METHOD PRIVATE M_Manual_Cylinder
VAR_INPUT
END_VAR
CylinderManualCtrl[1](bTrigger:=StorageManualCommand.UpCV.FeedInPress1.Exetend);
CylinderManualCtrl[2](bTrigger:=StorageManualCommand.UpCV.FeedInPress2.Exetend);
CylinderManualCtrl[3](bTrigger:=StorageManualCommand.UpCV.DiameterPress.Exetend);
CylinderManualCtrl[4](bTrigger:=StorageManualCommand.UpCV.CamaraPress1.Exetend);
CylinderManualCtrl[5](bTrigger:=StorageManualCommand.UpCV.CamaraPress2.Exetend);
CylinderManualCtrl[6](bTrigger:=StorageManualCommand.UpCV.CamaraPress3.Exetend);
CylinderManualCtrl[7](bTrigger:=StorageManualCommand.UpCV.CamaraPress4.Exetend);
CylinderManualCtrl[8](bTrigger:=StorageManualCommand.UpCV.Block1.Exetend);
CylinderManualCtrl[9](bTrigger:=StorageManualCommand.UpCV.Block2.Exetend);
CylinderManualCtrl[10](bTrigger:=StorageManualCommand.UpCV.Block3.Exetend);
CylinderManualCtrl[11](bTrigger:=StorageManualCommand.UpCV.DiameterHoriz.Exetend);
CylinderManualCtrl[12](bTrigger:=StorageManualCommand.UpCV.DiameterVert.Exetend);
CylinderManualCtrl[13](bTrigger:=StorageManualCommand.UpCV.DiameterClamp.Exetend);
CylinderManualCtrl[14](bTrigger:=StorageManualCommand.UpCV.StackPush.Exetend);
CylinderManualCtrl[15](bTrigger:=AllocateManualCommand.PullOutCV.AsidePress1.Exetend);
CylinderManualCtrl[16](bTrigger:=AllocateManualCommand.PullOutCV.AsidePress2.Exetend);
CylinderManualCtrl[17](bTrigger:=AllocateManualCommand.PullOutCV.AsideBlock.Exetend);
CylinderManualCtrl[18](bTrigger:=AllocateManualCommand.PullOutCV.BsidePress1.Exetend);
CylinderManualCtrl[19](bTrigger:=AllocateManualCommand.PullOutCV.BsidePress2.Exetend);
CylinderManualCtrl[20](bTrigger:=AllocateManualCommand. PullOutCV.BsideBlock.Exetend);
CylinderManualCtrl[21](bTrigger:=StorageManualCommand.LowCV.Press1.Exetend);
CylinderManualCtrl[22](bTrigger:=StorageManualCommand.LowCV.Press2.Exetend);
CylinderManualCtrl[23](bTrigger:=StorageManualCommand.LowCV.Press3.Exetend);
CylinderManualCtrl[24](bTrigger:=StorageManualCommand.LowCV.Press4.Exetend);
CylinderManualCtrl[25](bTrigger:=StorageManualCommand.LowCV.Block1.Exetend);
CylinderManualCtrl[26](bTrigger:=StorageManualCommand.LowCV.Block2.Exetend);
CylinderManualCtrl[27](bTrigger:=AllocateManualCommand.AllocatedRobot.LeftVert1.Exetend);
CylinderManualCtrl[28](bTrigger:=AllocateManualCommand.AllocatedRobot.LeftVert2.Exetend);
CylinderManualCtrl[29](bTrigger:=AllocateManualCommand.AllocatedRobot.RightVert1.Exetend);
CylinderManualCtrl[30](bTrigger:=AllocateManualCommand.AllocatedRobot.RightVert2.Exetend);
CylinderManualCtrl[31](bTrigger:=AllocateManualCommand.AllocatedRobot.LeftClamp1.Exetend);
CylinderManualCtrl[32](bTrigger:=AllocateManualCommand.AllocatedRobot.LeftClamp2.Exetend);
CylinderManualCtrl[33](bTrigger:=AllocateManualCommand.AllocatedRobot.RightClamp1.Exetend);
CylinderManualCtrl[34](bTrigger:=AllocateManualCommand.AllocatedRobot.RightClamp2.Exetend);
CylinderManualCtrl[35](bTrigger:=AllocateManualCommand.RoundBelt.WorkZone_Press.Exetend);
CylinderManualCtrl[36](bTrigger:=AllocateManualCommand.RoundBelt.WorkZone_Plug.Exetend);
CylinderManualCtrl[37](bTrigger:=AllocateManualCommand.RoundBelt.ChargeZone_Plug.Exetend);
CylinderManualCtrl[38](bTrigger:=AllocateManualCommand.RoundBelt.TransmitCVZone_Plug.Exetend);
CylinderManualCtrl[39](bTrigger:=AllocateManualCommand.OutRobot.AsideVert.Exetend);
CylinderManualCtrl[40](bTrigger:=AllocateManualCommand.OutRobot.BsideVert.Exetend);
CylinderManualCtrl[41](bTrigger:=AllocateManualCommand.OutRobot.AsideClamp.Exetend);
CylinderManualCtrl[42](bTrigger:=AllocateManualCommand.OutRobot.BsideClamp.Exetend);
CylinderManualCtrl[43](bTrigger:=AllocateManualCommand.TransCV.CamaraHoriz .Exetend);
CylinderManualCtrl[44](bTrigger:=AllocateManualCommand.TransCV.DifferentSizeCV_Press2.Exetend);
CylinderManualCtrl[45](bTrigger:=AllocateManualCommand.TransCV.DifferentSizeCV_Press1.Exetend);
CylinderManualCtrl[46](bTrigger:=AllocateManualCommand.TransCV.DifferentSizeCV_Block1.Exetend);
CylinderManualCtrl[47](bTrigger:=AllocateManualCommand.TransCV.SameSizeCV_Press4.Exetend);
CylinderManualCtrl[48](bTrigger:=AllocateManualCommand.TransCV.SameSizeCV_Press3.Exetend);
CylinderManualCtrl[49](bTrigger:=AllocateManualCommand.TransCV.SameSizeCV_Press2.Exetend);
CylinderManualCtrl[50](bTrigger:=AllocateManualCommand.TransCV.SameSizeCV_Press1.Exetend);
CylinderManualCtrl[51](bTrigger:=AllocateManualCommand.TransCV.SameSizeCV_Block2.Exetend);
CylinderManualCtrl[52](bTrigger:=AllocateManualCommand.TransCV.SameSizeCV_Block1 .Exetend);
CylinderManualCtrl[53](bTrigger:=AllocateManualCommand.TurnTable.Press.Exetend);
END_METHOD

METHOD PRIVATE M_Manual_Motor
VAR_INPUT
END_VAR
/////////////////////////   WareHous A
MotorManualCtrl[1](bForward	:=StorageManualCommand.WareHouseCV_01.Forward	);
MotorManualCtrl[2](bForward	:=StorageManualCommand.WareHouseCV_02.Forward	);
MotorManualCtrl[3](bForward	:=StorageManualCommand.WareHouseCV_03.Forward	);
MotorManualCtrl[4](bForward	:=StorageManualCommand.WareHouseCV_04.Forward	);
MotorManualCtrl[5](bForward	:=StorageManualCommand.WareHouseCV_05.Forward	);
MotorManualCtrl[6](bForward	:=StorageManualCommand.WareHouseCV_06.Forward	);
MotorManualCtrl[7](bForward	:=StorageManualCommand.WareHouseCV_07.Forward	);
MotorManualCtrl[8](bForward	:=StorageManualCommand.WareHouseCV_08.Forward	);
MotorManualCtrl[9](bForward	:=StorageManualCommand.WareHouseCV_09.Forward	);
MotorManualCtrl[10](bForward:=StorageManualCommand.WareHouseCV_10.Forward	);
MotorManualCtrl[11](bForward:=StorageManualCommand.WareHouseCV_11.Forward	);
MotorManualCtrl[12](bForward:=StorageManualCommand.WareHouseCV_12.Forward	);
MotorManualCtrl[13](bForward:=StorageManualCommand.WareHouseCV_13.Forward	);
MotorManualCtrl[14](bForward:=StorageManualCommand.WareHouseCV_14.Forward	);
MotorManualCtrl[15](bForward:=StorageManualCommand.WareHouseCV_15.Forward	);
MotorManualCtrl[16](bForward:=StorageManualCommand.WareHouseCV_16.Forward	);
MotorManualCtrl[17](bForward:=StorageManualCommand.WareHouseCV_17.Forward	);
MotorManualCtrl[18](bForward:=StorageManualCommand.WareHouseCV_18.Forward	);
MotorManualCtrl[19](bForward:=StorageManualCommand.WareHouseCV_19.Forward	);
MotorManualCtrl[20](bForward:=StorageManualCommand.WareHouseCV_20.Forward	);
MotorManualCtrl[21](bForward:=StorageManualCommand.UpCV.UpCV.Forward	);
MotorManualCtrl[22](bForward:=StorageManualCommand.LowCV.LowCV.Forward	);

MotorManualCtrl[23](bForward:=AllocateManualCommand.PullOutCV.PullOutCV_A.Forward);
MotorManualCtrl[24](bForward:=AllocateManualCommand.PullOutCV.PullOutCV_B.Forward);
MotorManualCtrl[25](bForward:=AllocateManualCommand.TransCV.TransmitSameSideCV.Forward);
MotorManualCtrl[26](bForward:=AllocateManualCommand.TransCV.TransmitDifferentSideCV.Forward);


MotorManualCtrl[1](bBackward	:=StorageManualCommand.WareHouseCV_10.Backward	);
MotorManualCtrl[2](bBackward	:=StorageManualCommand.WareHouseCV_09.Backward	);
MotorManualCtrl[3](bBackward	:=StorageManualCommand.WareHouseCV_08.Backward	);
MotorManualCtrl[4](bBackward	:=StorageManualCommand.WareHouseCV_07.Backward	);
MotorManualCtrl[5](bBackward	:=StorageManualCommand.WareHouseCV_06.Backward	);
MotorManualCtrl[6](bBackward	:=StorageManualCommand.WareHouseCV_05.Backward	);
MotorManualCtrl[7](bBackward	:=StorageManualCommand.WareHouseCV_04.Backward	);
MotorManualCtrl[8](bBackward	:=StorageManualCommand.WareHouseCV_03.Backward	);
MotorManualCtrl[9](bBackward	:=StorageManualCommand.WareHouseCV_02.Backward	);
MotorManualCtrl[10](bBackward:=StorageManualCommand.WareHouseCV_01.Backward	);
MotorManualCtrl[11](bBackward:=StorageManualCommand.WareHouseCV_20.Backward	);
MotorManualCtrl[12](bBackward:=StorageManualCommand.WareHouseCV_19.Backward	);
MotorManualCtrl[13](bBackward:=StorageManualCommand.WareHouseCV_18.Backward	);
MotorManualCtrl[14](bBackward:=StorageManualCommand.WareHouseCV_17.Backward	);
MotorManualCtrl[15](bBackward:=StorageManualCommand.WareHouseCV_16.Backward	);
MotorManualCtrl[16](bBackward:=StorageManualCommand.WareHouseCV_15.Backward	);
MotorManualCtrl[17](bBackward:=StorageManualCommand.WareHouseCV_14.Backward	);
MotorManualCtrl[18](bBackward:=StorageManualCommand.WareHouseCV_13.Backward	);
MotorManualCtrl[19](bBackward:=StorageManualCommand.WareHouseCV_12.Backward	);
MotorManualCtrl[20](bBackward:=StorageManualCommand.WareHouseCV_11.Backward	);
MotorManualCtrl[21](bBackward:=StorageManualCommand.UpCV.UpCV.Backward	);
MotorManualCtrl[22](bBackward:=StorageManualCommand.LowCV.LowCV.Backward	);

MotorManualCtrl[23](bBackward:=AllocateManualCommand.PullOutCV.PullOutCV_A.Backward);
MotorManualCtrl[24](bBackward:=AllocateManualCommand.PullOutCV.PullOutCV_B.Backward);
MotorManualCtrl[25](bBackward:=AllocateManualCommand.TransCV.TransmitSameSideCV.Backward);
MotorManualCtrl[26](bBackward:=AllocateManualCommand.TransCV.TransmitDifferentSideCV.Backward);

MotorManualCtrl[1](bStop	:=StorageManualCommand.WareHouseCV_10.Stopped	);
MotorManualCtrl[2](bStop	:=StorageManualCommand.WareHouseCV_09.Stopped	);
MotorManualCtrl[3](bStop	:=StorageManualCommand.WareHouseCV_08.Stopped	);
MotorManualCtrl[4](bStop	:=StorageManualCommand.WareHouseCV_07.Stopped	);
MotorManualCtrl[5](bStop	:=StorageManualCommand.WareHouseCV_06.Stopped	);
MotorManualCtrl[6](bStop	:=StorageManualCommand.WareHouseCV_05.Stopped	);
MotorManualCtrl[7](bStop	:=StorageManualCommand.WareHouseCV_04.Stopped	);
MotorManualCtrl[8](bStop	:=StorageManualCommand.WareHouseCV_03.Stopped	);
MotorManualCtrl[9](bStop	:=StorageManualCommand.WareHouseCV_02.Stopped	);
MotorManualCtrl[10](bStop:=StorageManualCommand.WareHouseCV_01.Stopped	);
MotorManualCtrl[11](bStop:=StorageManualCommand.WareHouseCV_20.Stopped	);
MotorManualCtrl[12](bStop:=StorageManualCommand.WareHouseCV_19.Stopped	);
MotorManualCtrl[13](bStop:=StorageManualCommand.WareHouseCV_18.Stopped	);
MotorManualCtrl[14](bStop:=StorageManualCommand.WareHouseCV_17.Stopped	);
MotorManualCtrl[15](bStop:=StorageManualCommand.WareHouseCV_16.Stopped	);
MotorManualCtrl[16](bStop:=StorageManualCommand.WareHouseCV_15.Stopped	);
MotorManualCtrl[17](bStop:=StorageManualCommand.WareHouseCV_14.Stopped	);
MotorManualCtrl[18](bStop:=StorageManualCommand.WareHouseCV_13.Stopped	);
MotorManualCtrl[19](bStop:=StorageManualCommand.WareHouseCV_12.Stopped	);
MotorManualCtrl[20](bStop:=StorageManualCommand.WareHouseCV_11.Stopped	);
MotorManualCtrl[21](bStop:=StorageManualCommand.UpCV.UpCV.Stopped	);
MotorManualCtrl[22](bStop:=StorageManualCommand.LowCV.LowCV.Stopped	);

MotorManualCtrl[23](bStop:=AllocateManualCommand.PullOutCV.PullOutCV_A.Stopped);
MotorManualCtrl[24](bStop:=AllocateManualCommand.PullOutCV.PullOutCV_B.Stopped);
MotorManualCtrl[25](bStop:=AllocateManualCommand.TransCV.TransmitSameSideCV.Stopped);
MotorManualCtrl[26](bStop:=AllocateManualCommand.TransCV.TransmitDifferentSideCV.Stopped);

(*IF StorageManualCommand.WareHouseCV_10.Forward THEN
    Motor.List.WareHouseCV_10.M_MoveForward());
ELSIF StorageManualCommand.WareHouseCV_10.Backward THEN
    Motor.List.WareHouseCV_10.M_MoveBackward());
ELSIF
    StorageManualCommand.WareHouseCV_10.Stopped OR NOT (StorageManualCommand.WareHouseCV_10.Forward OR StorageManualCommand.WareHouseCV_10.Backward)
    THEN
    Motor.List.WareHouseCV_10.M_MotorStop());
END_IF

IF StorageManualCommand.WareHouseCV_09.Forward THEN
    Motor.List.WareHouseCV_09.M_MoveForward());
ELSIF StorageManualCommand.WareHouseCV_09.Backward THEN
    Motor.List.WareHouseCV_09.M_MoveBackward());
ELSIF StorageManualCommand.WareHouseCV_09.Stopped OR NOT (StorageManualCommand.WareHouseCV_09.Forward OR StorageManualCommand.WareHouseCV_09.Backward)
    THEN
    Motor.List.WareHouseCV_09.M_MotorStop());
END_IF

IF StorageManualCommand.WareHouseCV_08.Forward THEN
    Motor.List.WareHouseCV_08.M_MoveForward());
ELSIF StorageManualCommand.WareHouseCV_08.Backward THEN
    Motor.List.WareHouseCV_08.M_MoveBackward());
ELSIF StorageManualCommand.WareHouseCV_08.Stopped OR NOT (StorageManualCommand.WareHouseCV_08.Forward OR StorageManualCommand.WareHouseCV_08.Backward)
    THEN
    Motor.List.WareHouseCV_08.M_MotorStop());
END_IF

IF StorageManualCommand.WareHouseCV_07.Forward THEN
    Motor.List.WareHouseCV_07.M_MoveForward());
ELSIF StorageManualCommand.WareHouseCV_07.Backward THEN
    Motor.List.WareHouseCV_07.M_MoveBackward());
ELSIF StorageManualCommand.WareHouseCV_07.Stopped OR NOT (StorageManualCommand.WareHouseCV_07.Forward OR StorageManualCommand.WareHouseCV_07.Backward)
    THEN
    Motor.List.WareHouseCV_07.M_MotorStop());
END_IF

IF StorageManualCommand.WareHouseCV_06.Forward THEN
    Motor.List.WareHouseCV_06.M_MoveForward());
ELSIF StorageManualCommand.WareHouseCV_06.Backward THEN
    Motor.List.WareHouseCV_06.M_MoveBackward());
ELSIF StorageManualCommand.WareHouseCV_06.Stopped OR NOT (StorageManualCommand.WareHouseCV_06.Forward OR StorageManualCommand.WareHouseCV_06.Backward)
    THEN
    Motor.List.WareHouseCV_06.M_MotorStop());
END_IF

IF StorageManualCommand.WareHouseCV_05.Forward THEN
    Motor.List.WareHouseCV_05.M_MoveForward());
ELSIF StorageManualCommand.WareHouseCV_05.Backward THEN
    Motor.List.WareHouseCV_05.M_MoveBackward());
ELSIF StorageManualCommand.WareHouseCV_05.Stopped OR NOT (StorageManualCommand.WareHouseCV_05.Forward OR StorageManualCommand.WareHouseCV_05.Backward)
    THEN
    Motor.List.WareHouseCV_05.M_MotorStop());
END_IF

IF StorageManualCommand.WareHouseCV_04.Forward THEN
    Motor.List.WareHouseCV_04.M_MoveForward());
ELSIF StorageManualCommand.WareHouseCV_04.Backward THEN
    Motor.List.WareHouseCV_04.M_MoveBackward());
ELSIF StorageManualCommand.WareHouseCV_04.Stopped OR NOT (StorageManualCommand.WareHouseCV_04.Forward OR StorageManualCommand.WareHouseCV_04.Backward)
    THEN
    Motor.List.WareHouseCV_04.M_MotorStop());
END_IF

IF StorageManualCommand.WareHouseCV_03.Forward THEN
    Motor.List.WareHouseCV_03.M_MoveForward());
ELSIF StorageManualCommand.WareHouseCV_03.Backward THEN
    Motor.List.WareHouseCV_03.M_MoveBackward());
ELSIF StorageManualCommand.WareHouseCV_03.Stopped OR NOT (StorageManualCommand.WareHouseCV_03.Forward OR StorageManualCommand.WareHouseCV_03.Backward)
    THEN
    Motor.List.WareHouseCV_03.M_MotorStop());
END_IF

IF StorageManualCommand.WareHouseCV_02.Forward THEN
    Motor.List.WareHouseCV_02.M_MoveForward());
ELSIF StorageManualCommand.WareHouseCV_02.Backward THEN
    Motor.List.WareHouseCV_02.M_MoveBackward());
ELSIF StorageManualCommand.WareHouseCV_02.Stopped OR NOT (StorageManualCommand.WareHouseCV_02.Forward OR StorageManualCommand.WareHouseCV_02.Backward)
    THEN
    Motor.List.WareHouseCV_02.M_MotorStop());
END_IF

IF StorageManualCommand.WareHouseCV_01.Forward THEN
    Motor.List.WareHouseCV_01.M_MoveForward());
ELSIF StorageManualCommand.WareHouseCV_01.Backward THEN
    Motor.List.WareHouseCV_01.M_MoveBackward());
ELSIF StorageManualCommand.WareHouseCV_01.Stopped OR NOT (StorageManualCommand.WareHouseCV_01.Forward OR StorageManualCommand.WareHouseCV_01.Backward)
    THEN
    Motor.List.WareHouseCV_01.M_MotorStop());
END_IF

///////////////////////      Warehouse B
IF StorageManualCommand.WareHouseCV_11.Forward THEN
    Motor.List.WareHouseCV_11.M_MoveForward());
ELSIF StorageManualCommand.WareHouseCV_11.Backward THEN
    Motor.List.WareHouseCV_11.M_MoveBackward());
ELSIF StorageManualCommand.WareHouseCV_11.Stopped OR NOT (StorageManualCommand.WareHouseCV_11.Forward OR StorageManualCommand.WareHouseCV_11.Backward)
    THEN
    Motor.List.WareHouseCV_11.M_MotorStop());
END_IF

IF StorageManualCommand.WareHouseCV_12.Forward THEN
    Motor.List.WareHouseCV_12.M_MoveForward());
ELSIF StorageManualCommand.WareHouseCV_12.Backward THEN
    Motor.List.WareHouseCV_12.M_MoveBackward());
ELSIF StorageManualCommand.WareHouseCV_12.Stopped OR NOT (StorageManualCommand.WareHouseCV_12.Forward OR StorageManualCommand.WareHouseCV_12.Backward)
    THEN
    Motor.List.WareHouseCV_12.M_MotorStop());
END_IF

IF StorageManualCommand.WareHouseCV_13.Forward THEN
    Motor.List.WareHouseCV_13.M_MoveForward());
ELSIF StorageManualCommand.WareHouseCV_13.Backward THEN
    Motor.List.WareHouseCV_13.M_MoveBackward());
ELSIF StorageManualCommand.WareHouseCV_13.Stopped OR NOT (StorageManualCommand.WareHouseCV_13.Forward OR StorageManualCommand.WareHouseCV_13.Backward)
    THEN
    Motor.List.WareHouseCV_13.M_MotorStop());
END_IF

IF StorageManualCommand.WareHouseCV_14.Forward THEN
    Motor.List.WareHouseCV_14.M_MoveForward());
ELSIF StorageManualCommand.WareHouseCV_14.Backward THEN
    Motor.List.WareHouseCV_14.M_MoveBackward());
ELSIF StorageManualCommand.WareHouseCV_14.Stopped OR NOT (StorageManualCommand.WareHouseCV_14.Forward OR StorageManualCommand.WareHouseCV_14.Backward)
    THEN
    Motor.List.WareHouseCV_14.M_MotorStop());
END_IF

IF StorageManualCommand.WareHouseCV_15.Forward THEN
    Motor.List.WareHouseCV_15.M_MoveForward());
ELSIF StorageManualCommand.WareHouseCV_15.Backward THEN
    Motor.List.WareHouseCV_15.M_MoveBackward());
ELSIF StorageManualCommand.WareHouseCV_15.Stopped OR NOT (StorageManualCommand.WareHouseCV_15.Forward OR StorageManualCommand.WareHouseCV_15.Backward)
    THEN
    Motor.List.WareHouseCV_15.M_MotorStop());
END_IF

IF StorageManualCommand.WareHouseCV_16.Forward THEN
    Motor.List.WareHouseCV_16.M_MoveForward());
ELSIF StorageManualCommand.WareHouseCV_16.Backward THEN
    Motor.List.WareHouseCV_16.M_MoveBackward());
ELSIF StorageManualCommand.WareHouseCV_16.Stopped OR NOT (StorageManualCommand.WareHouseCV_16.Forward OR StorageManualCommand.WareHouseCV_16.Backward)
    THEN
    Motor.List.WareHouseCV_16.M_MotorStop());
END_IF

IF StorageManualCommand.WareHouseCV_17.Forward THEN
    Motor.List.WareHouseCV_17.M_MoveForward());
ELSIF StorageManualCommand.WareHouseCV_17.Backward THEN
    Motor.List.WareHouseCV_17.M_MoveBackward());
ELSIF StorageManualCommand.WareHouseCV_17.Stopped OR NOT (StorageManualCommand.WareHouseCV_17.Forward OR StorageManualCommand.WareHouseCV_17.Backward)
    THEN
    Motor.List.WareHouseCV_17.M_MotorStop());
END_IF

IF StorageManualCommand.WareHouseCV_18.Forward THEN
    Motor.List.WareHouseCV_18.M_MoveForward());
ELSIF StorageManualCommand.WareHouseCV_18.Backward THEN
    Motor.List.WareHouseCV_18.M_MoveBackward());
ELSIF StorageManualCommand.WareHouseCV_18.Stopped OR NOT (StorageManualCommand.WareHouseCV_18.Forward OR StorageManualCommand.WareHouseCV_18.Backward)
    THEN
    Motor.List.WareHouseCV_18.M_MotorStop());
END_IF

IF StorageManualCommand.WareHouseCV_19.Forward THEN
    Motor.List.WareHouseCV_19.M_MoveForward());
ELSIF StorageManualCommand.WareHouseCV_19.Backward THEN
    Motor.List.WareHouseCV_19.M_MoveBackward());
ELSIF StorageManualCommand.WareHouseCV_19.Stopped OR NOT (StorageManualCommand.WareHouseCV_19.Forward OR StorageManualCommand.WareHouseCV_19.Backward)
    THEN
    Motor.List.WareHouseCV_19.M_MotorStop());
END_IF

IF StorageManualCommand.WareHouseCV_20.Forward THEN
    Motor.List.WareHouseCV_20.M_MoveForward());
ELSIF StorageManualCommand.WareHouseCV_20.Backward THEN
    Motor.List.WareHouseCV_20.M_MoveBackward());
ELSIF StorageManualCommand.WareHouseCV_20.Stopped OR NOT (StorageManualCommand.WareHouseCV_20.Forward OR StorageManualCommand.WareHouseCV_20.Backward)
    THEN
    Motor.List.WareHouseCV_20.M_MotorStop());
END_IF

///////////////////////////////////   TransCV
IF AllocateManualCommand.TransCV.TransmitSameSideCV.Forward THEN
    Motor.List.TransmitSameSideCV.M_MoveForward());
ELSIF AllocateManualCommand.TransCV.TransmitSameSideCV.Backward THEN
    Motor.List.TransmitSameSideCV.M_MoveBackward());
ELSIF AllocateManualCommand.TransCV.TransmitSameSideCV.Stopped OR NOT 
	(AllocateManualCommand.TransCV.TransmitSameSideCV.Forward OR AllocateManualCommand.TransCV.TransmitSameSideCV.Backward) THEN
    Motor.List.TransmitSameSideCV.M_MotorStop());
END_IF

IF AllocateManualCommand.TransCV.TransmitDifferentSideCV.Forward THEN
    Motor.List.TransmitDifferentSideCV.M_MoveForward());
ELSIF AllocateManualCommand.TransCV.TransmitDifferentSideCV.Backward THEN
    Motor.List.TransmitDifferentSideCV.M_MoveBackward());
ELSIF AllocateManualCommand.TransCV.TransmitDifferentSideCV.Stopped OR NOT 
	(AllocateManualCommand.TransCV.TransmitDifferentSideCV.Forward OR AllocateManualCommand.TransCV.TransmitDifferentSideCV.Backward) THEN
    Motor.List.TransmitDifferentSideCV.M_MotorStop());
END_IF

//////////////////////////////////////   PullOutCV
IF AllocateManualCommand.PullOutCV.PullOutCV_A.Forward THEN
    Motor.List.PullOutCV_A.M_MoveForward());
ELSIF AllocateManualCommand.PullOutCV.PullOutCV_A.Backward THEN
    Motor.List.PullOutCV_A.M_MoveBackward());
ELSIF AllocateManualCommand.PullOutCV.PullOutCV_A.Stopped OR NOT
	(AllocateManualCommand.PullOutCV.PullOutCV_A.Forward OR AllocateManualCommand.PullOutCV.PullOutCV_A.Backward) THEN
    Motor.List.PullOutCV_A.M_MotorStop());
END_IF

IF AllocateManualCommand.PullOutCV.PullOutCV_B.Forward THEN
    Motor.List.PullOutCV_B.M_MoveForward());
ELSIF AllocateManualCommand.PullOutCV.PullOutCV_B.Backward THEN
    Motor.List.PullOutCV_B.M_MoveBackward());
ELSIF AllocateManualCommand.PullOutCV.PullOutCV_B.Stopped OR NOT 
	(AllocateManualCommand.PullOutCV.PullOutCV_B.Forward OR AllocateManualCommand.PullOutCV.PullOutCV_B.Backward) THEN
    Motor.List.PullOutCV_B.M_MotorStop());
END_IF

////////////////////////////////////////    Upper & Lower CV
IF StorageManualCommand.UpCV.UpCV.Forward THEN
    Motor.List.UpCV.M_MoveForward());
ELSIF StorageManualCommand.UpCV.UpCV.Backward THEN
    Motor.List.UpCV.M_MoveBackward());
ELSIF StorageManualCommand.UpCV.UpCV.Stopped OR NOT 
	(StorageManualCommand.UpCV.UpCV.Forward OR StorageManualCommand.UpCV.UpCV.Backward) THEN
    Motor.List.UpCV.M_MotorStop());
END_IF

IF StorageManualCommand.LowCV.LowCV.Forward THEN
    Motor.List.LowCV.M_MoveForward());
ELSIF StorageManualCommand.LowCV.LowCV.Backward THEN
    Motor.List.LowCV.M_MoveBackward());
ELSIF StorageManualCommand.LowCV.LowCV.Stopped OR NOT 
	(StorageManualCommand.LowCV.LowCV.Forward OR StorageManualCommand.LowCV.LowCV.Backward) THEN
    Motor.List.LowCV.M_MotorStop());
END_IF
*)
END_METHOD

METHOD M_ManualAllocateHoming
VAR_INPUT
END_VAR
//fbAllocateArea.fbAllocateHome.xExecute := Service_Handshake.AllocationRegionHome.HandShake.Execute;
IF Service_Handshake.AllocationRegionHome.HandShake.Execute THEN
	fbAllocateArea.M_StartHoming();
END_IF
Service_Handshake.AllocationRegionHome.HandShake.Busy := fbAllocateArea.fbAllocateHome.xBusy;
Service_Handshake.AllocationRegionHome.HandShake.Done := fbAllocateArea.fbAllocateHome.xDone;
Service_Handshake.AllocationRegionHome.HandShake.Error := fbAllocateArea.fbAllocateHome.xError;
IF  NOT Service_Handshake.AllocationRegionHome.HandShake.Execute THEN
	fbAllocateArea.M_StopHoming();
END_IF

Service_Handshake.AllocationRegionHome.Homed := fbAllocateArea.Homed;
END_METHOD

METHOD PRIVATE M_ManualMachineHome
VAR_INPUT
END_VAR
IF Service_Handshake.MachineHome.HandShake.Execute THEN
	M_StartHoming();
END_IF
Service_Handshake.MachineHome.HandShake.Busy := fbMachineHoming.xBusy;
Service_Handshake.MachineHome.HandShake.Done  := fbMachineHoming.xDone;
Service_Handshake.MachineHome.HandShake.Error := fbMachineHoming.xError;
IF NOT Service_Handshake.MachineHome.HandShake.Execute THEN
	M_StopHoming();
END_IF

Service_Handshake.MachineHome.Homed := MachineHomed;
END_METHOD

METHOD M_ManualShippingHoming 
VAR_INPUT
END_VAR
//fbStorageArea.fbStoragehoming.xExecute := Service_Handshake.StorageRegionHome.HandShake.Execute;
IF Service_Handshake.FGARegionHome.HandShake.Execute THEN
	fbShippingArea.M_StartHoming();
END_IF
Service_Handshake.FGARegionHome.HandShake.Busy := fbShippingArea.fbshippinghoming.xBusy;
Service_Handshake.FGARegionHome.HandShake.Done := fbShippingArea.fbshippinghoming.xDone;
Service_Handshake.FGARegionHome.HandShake.Error := fbShippingArea.fbshippinghoming.xError;
IF NOT Service_Handshake.FGARegionHome.HandShake.Execute  THEN
	fbShippingArea.M_StopHoming();
END_IF

Service_Handshake.FGARegionHome.Homed := fbShippingArea.Homed;
END_METHOD

METHOD M_ManualStorageHoming
VAR_INPUT
END_VAR
//fbStorageArea.fbStoragehoming.xExecute := Service_Handshake.StorageRegionHome.HandShake.Execute;
IF Service_Handshake.StorageRegionHome.HandShake.Execute THEN
	fbStorageArea.M_StartHoming();
END_IF
Service_Handshake.StorageRegionHome.HandShake.Busy := fbStorageArea.fbStoragehoming.xBusy;
Service_Handshake.StorageRegionHome.HandShake.Done := fbStorageArea.fbStoragehoming.xDone;
Service_Handshake.StorageRegionHome.HandShake.Error := fbStorageArea.fbStoragehoming.xError;
IF  NOT Service_Handshake.StorageRegionHome.HandShake.Execute THEN
	fbStorageArea.M_StopHoming();
END_IF

Service_Handshake.StorageRegionHome.Homed := fbStorageArea.Homed;
END_METHOD

METHOD M_Resetting
VAR
	CylinderIndex : INT;
	MotorIndex : INT;
END_VAR
FOR CylinderIndex := 1 TO 53 DO
	fbAllocateArea.M_TransCVCameraPress_ManualMode();
    Cylinder.arCylinder[CylinderIndex].xEnable := TRUE;
	CylinderManualCtrl[CylinderIndex].Cylinder REF= Cylinder.arCylinder[CylinderIndex];
END_FOR

FOR CylinderIndex := 1 TO 53 DO
    Cylinder.arCylinder[CylinderIndex].EnableSimulation := EnableSimulation;
END_FOR

FOR MotorIndex := 1 TO 26 DO
    Motor.arMotor[MotorIndex].xEnable := TRUE;
	MotorManualCtrl[MotorIndex].Motor REF= Motor.arMotor[MotorIndex];
END_FOR

// Reference 
ReferenceHMI();
RefStorageService();
RefAllocateService();
RefShippingService();

// State control
GVL_Machine.PackTags[UnitNo.Allocate].Command.CntrlCmd := ePMLCommand_Reset;
GVL_Machine.PackTags[UnitNo.Storage].Command.CntrlCmd := ePMLCommand_Reset;
GVL_Machine.PackTags[UnitNo.Shipping].Command.CntrlCmd := ePMLCommand_Reset;
arAxisCtrl_gb[AxisNo.RoundBelt].Admin.PositionType := E_PositionType.Modulo;
arAxisCtrl_gb[AxisNo.TurnTable].Admin.PositionType := E_PositionType.Modulo;

CASE eModeCurrent OF
    E_UnitMode.Manual:
        IF GVL_Machine.PackTags[UnitNo.Allocate].Status.StateCurrent = ePMLState_Idle AND
            GVL_Machine.PackTags[UnitNo.Storage].Status.StateCurrent = ePMLState_Idle AND
            GVL_Machine.PackTags[UnitNo.Shipping].Status.StateCurrent = ePMLState_Idle //
			 THEN
            M_StateComplete();
        END_IF
		IF ErrorTableInitDone THEN
			M_General_AlarmRegister();
		END_IF
    E_UnitMode.Auto:
        IF GVL_Machine.PackTags[UnitNo.Allocate].Status.StateCurrent = ePMLState_Idle AND
            GVL_Machine.PackTags[UnitNo.Storage].Status.StateCurrent = ePMLState_Idle AND
            GVL_Machine.PackTags[UnitNo.Shipping].Status.StateCurrent = ePMLState_Idle //AND
             THEN
            M_StateComplete();
        END_IF
		IF ErrorTableInitDone THEN
			M_General_AlarmRegister();
		END_IF
END_CASE
END_METHOD

METHOD M_StartHoming
VAR_INPUT
END_VAR
fbMachineHoming.xExecute := TRUE;
END_METHOD

METHOD M_Starting
// State control
GVL_Machine.PackTags[UnitNo.Allocate].Command.CntrlCmd := ePMLCommand_Start;
GVL_Machine.PackTags[UnitNo.Storage].Command.CntrlCmd := ePMLCommand_Start;
GVL_Machine.PackTags[UnitNo.Shipping].Command.CntrlCmd := ePMLCommand_Start;

CASE eModeCurrent OF
    E_UnitMode.Manual, E_UnitMode.Auto:
        IF GVL_Machine.PackTags[UnitNo.Allocate].Status.StateCurrent = ePMLState_Execute AND
            GVL_Machine.PackTags[UnitNo.Allocate].Status.StateCurrent = ePMLState_Execute AND
            GVL_Machine.PackTags[UnitNo.Allocate].Status.StateCurrent = ePMLState_Execute THEN
            M_StateComplete();
        END_IF
END_CASE
END_METHOD

METHOD M_StopHoming
VAR_INPUT
END_VAR
fbMachineHoming.xExecute := FALSE;
END_METHOD

METHOD M_Stopped
VAR
	CylinderIndex : INT;
	MotorIndex : INT;
	ServoIndex : INT;
END_VAR
FOR ServoIndex := 1 TO 7 DO
	IF arAxisCtrl_gb[ServoIndex].Admin.Axis.Status.Error THEN
		arAxisCtrl_gb[ServoIndex].Admin.ClearError := FALSE;
	END_IF
END_FOR

IF eModeCurrent = E_UnitMode.Auto THEN
	GVL_Machine.PackTags[UnitNo.Storage].Command.UnitMode := E_UnitMode.Auto;
	GVL_Machine.PackTags[UnitNo.Allocate].Command.UnitMode := E_UnitMode.Auto;
	GVL_Machine.PackTags[UnitNo.Shipping].Command.UnitMode := E_UnitMode.Auto;
ELSIF eModeCurrent = E_UnitMode.Manual THEN
	GVL_Machine.PackTags[UnitNo.Storage].Command.UnitMode := E_UnitMode.Manual;
	GVL_Machine.PackTags[UnitNo.Allocate].Command.UnitMode := E_UnitMode.Manual;
	GVL_Machine.PackTags[UnitNo.Shipping].Command.UnitMode := E_UnitMode.Manual;
END_IF

CASE eModeCurrent OF
	E_UnitMode.Manual:
		IF GVL_Machine.PackTags[UnitNo.Allocate].Status.UnitModeCurrent = E_UnitMode.Manual AND 
			GVL_Machine.PackTags[UnitNo.Allocate].Status.StateCurrent = ePMLState_Stopped AND
			GVL_Machine.PackTags[UnitNo.Storage].Status.UnitModeCurrent = E_UnitMode.Manual AND 
			GVL_Machine.PackTags[UnitNo.Storage].Status.StateCurrent = ePMLState_Stopped AND
			GVL_Machine.PackTags[UnitNo.Shipping].Status.UnitModeCurrent = E_UnitMode.Manual AND 
			GVL_Machine.PackTags[UnitNo.Shipping].Status.StateCurrent = ePMLState_Stopped THEN
			M_StateComplete();
		END_IF
	E_UnitMode.Auto:
		IF GVL_Machine.PackTags[UnitNo.Allocate].Status.UnitModeCurrent = E_UnitMode.Auto AND 
			GVL_Machine.PackTags[UnitNo.Allocate].Status.StateCurrent = ePMLState_Stopped AND
			GVL_Machine.PackTags[UnitNo.Storage].Status.UnitModeCurrent = E_UnitMode.Auto AND 
			GVL_Machine.PackTags[UnitNo.Storage].Status.StateCurrent = ePMLState_Stopped AND
			GVL_Machine.PackTags[UnitNo.Shipping].Status.UnitModeCurrent = E_UnitMode.Auto AND 
			GVL_Machine.PackTags[UnitNo.Shipping].Status.StateCurrent = ePMLState_Stopped THEN
			M_StateComplete();
		END_IF
END_CASE
END_METHOD

METHOD M_Stopping
VAR
	CylinderIndex :INT;
	MotorIndex : INT;
END_VAR
CASE eModeCurrent OF
    E_UnitMode.Manual:
        GVL_Machine.PackTags[UnitNo.Allocate].Command.UnitMode := E_UnitMode.Manual;
        GVL_Machine.PackTags[UnitNo.Allocate].Command.CntrlCmd := ePMLCommand_Stop;
        GVL_Machine.PackTags[UnitNo.Storage].Command.UnitMode  := E_UnitMode.Manual;
        GVL_Machine.PackTags[UnitNo.Storage].Command.CntrlCmd  := ePMLCommand_Stop;
        GVL_Machine.PackTags[UnitNo.Shipping].Command.UnitMode := E_UnitMode.Manual;
        GVL_Machine.PackTags[UnitNo.Shipping].Command.CntrlCmd := ePMLCommand_Stop;
		FOR CylinderIndex := 1 TO 53 DO
			Cylinder.arCylinder[CylinderIndex].xEnable := FALSE;
		END_FOR
		FOR MotorIndex := 1 TO 26 DO
			Motor.arMotor[MotorIndex].xEnable := FALSE;
		END_FOR
		TableMove.xExecute := FALSE;
        IF GVL_Machine.PackTags[UnitNo.Allocate].Status.UnitModeCurrent = E_UnitMode.Manual AND
           GVL_Machine.PackTags[UnitNo.Allocate].Status.StateCurrent = ePMLState_Stopped AND
           GVL_Machine.PackTags[UnitNo.Storage].Status.UnitModeCurrent = E_UnitMode.Manual AND
           GVL_Machine.PackTags[UnitNo.Storage].Status.StateCurrent = ePMLState_Stopped AND
           GVL_Machine.PackTags[UnitNo.Shipping].Status.UnitModeCurrent = E_UnitMode.Manual AND
           GVL_Machine.PackTags[UnitNo.Shipping].Status.StateCurrent = ePMLState_Stopped AND NOT
		   TableMove.xError
            THEN
            M_StateComplete();
        END_IF
	E_UnitMode.Auto:
        GVL_Machine.PackTags[UnitNo.Allocate].Command.UnitMode := E_UnitMode.Auto;
        GVL_Machine.PackTags[UnitNo.Allocate].Command.CntrlCmd := ePMLCommand_Stop;
        GVL_Machine.PackTags[UnitNo.Storage].Command.UnitMode  := E_UnitMode.Auto;
        GVL_Machine.PackTags[UnitNo.Storage].Command.CntrlCmd  := ePMLCommand_Stop;
        GVL_Machine.PackTags[UnitNo.Shipping].Command.UnitMode := E_UnitMode.Auto;
        GVL_Machine.PackTags[UnitNo.Shipping].Command.CntrlCmd := ePMLCommand_Stop;
		FOR CylinderIndex := 1 TO 53 DO
			Cylinder.arCylinder[CylinderIndex].xEnable := FALSE;
		END_FOR
		FOR MotorIndex := 1 TO 26 DO
			Motor.arMotor[MotorIndex].xEnable := FALSE;
		END_FOR
		TableMove.xExecute := FALSE;
        IF GVL_Machine.PackTags[UnitNo.Allocate].Status.UnitModeCurrent = E_UnitMode.Auto AND
           GVL_Machine.PackTags[UnitNo.Allocate].Status.StateCurrent = ePMLState_Stopped AND
           GVL_Machine.PackTags[UnitNo.Storage].Status.UnitModeCurrent = E_UnitMode.Auto AND
           GVL_Machine.PackTags[UnitNo.Storage].Status.StateCurrent = ePMLState_Stopped AND
           GVL_Machine.PackTags[UnitNo.Shipping].Status.UnitModeCurrent = E_UnitMode.Auto AND
           GVL_Machine.PackTags[UnitNo.Shipping].Status.StateCurrent = ePMLState_Stopped AND NOT
		   TableMove.xError
            THEN
            M_StateComplete();
        END_IF
END_CASE
END_METHOD

METHOD PRIVATE M_StroageRobotSafeCheck : BOOL
VAR_INPUT
END_VAR
IF FanucRobot.List.StorageRobot._DI12.BzoneWaitAllow THEN
	IF NOT arAxisCtrl_gb[AxisNo.RoundBelt].Admin.Axis.Status.Moving
	    AND NOT fbAllocateArea.RoundBeltControl.xBusy
		AND NOT fbAllocateArea.RoundBeltControl.xError
		AND NOT fbAllocateArea.RoundBeltControl.xDone THEN
			FanucRobot.List.StorageRobot.Bzone_AllowWork := TRUE;
	END_IF
END_IF

IF NOT FanucRobot.List.StorageRobot._DI12.BzoneInWork 
	AND NOT FanucRobot.List.StorageRobot._DI12.BzoneWaitAllow THEN
	FanucRobot.List.StorageRobot.Bzone_AllowWork := FALSE	;
END_IF
END_METHOD

METHOD M_Suspended
M_StateComplete();
END_METHOD

METHOD M_Suspending
M_StateComplete();
END_METHOD

METHOD M_Undefined
CASE eModeCurrent OF
    E_UnitMode.Undefined:
		PackTag.Command.UnitMode := E_UnitMode.Manual;
		PackTag.Command.CntrlCmd := ePMLCommand_Abort;
		M_StateComplete();
END_CASE
END_METHOD

METHOD M_Unholding
M_StateComplete();
END_METHOD

METHOD M_Unsuspending
END_METHOD

METHOD PRIVATE RefAllocateService
VAR_INPUT
END_VAR
AllocateService.AllocateMoveStructure 				REF= Service_Handshake.AllocateMoveStructure;
AllocateService.AllocateCircleMove 					REF= Service_Handshake.AllocateCircleMove;
AllocateService.TurnTableMove 						REF= Service_Handshake.TurnTableMove;

// Allocating
AllocateService.AutoMode_AllocateBatchMode 			REF= Service_Handshake.AutoMode_AllocateBatchMode;
AllocateService.AutoMode_SimpleAllocation_Batch 	REF= Service_Handshake.AutoMode_SimpleAllocation_Batch;
AllocateService.AutoMode_AllocateBatchMode_Reverse  REF= Service_Handshake.AutoMode_AllocateBatchMode_Reverse;

//OutRobot
AllocateService.AutoMode_RareBoxMove 				REF= Service_Handshake.AutoMode_RareBoxMove;
AllocateService.AutoMode_EmptyBoxMove 				REF= Service_Handshake.AutoMode_EmptyBoxMove;
AllocateService.AutoMode_BoxMoveReverse 			REF= Service_Handshake.AutoMode_BoxMoveReverse;

//TransCV camera 
AllocateService.AutoMode_SameSizeCVCamera 			REF= Service_Handshake.AutoMode_SameSizeCVCamera;
AllocateService.AutoMode_DifferentCVCamera 			REF= Service_Handshake.AutoMode_DifferentCVCamera;

//AllocateArea Home
AllocateService.AllocateRegionHome					REF= Service_Handshake.AllocationRegionHome;

// Pullout 
AllocateService.AutoMode_PullOutConveyor 			REF= Service_Handshake.AutoMode_PullOutConveyor;

//AutoModeUse*-------自動模式圓帶單動
   AllocateService.AutoMode_AllocateCircleMove 		 REF= Service_Handshake.AutoMode_AllocateCircleMove;

 //AutoModeUse*-------圓盤移動
    AllocateService.AutoMode_TurnTableMOve  		REF= Service_Handshake.AutoMode_TurnTableMOve;
	
//Allocate robot move
AllocateService.AllocateRobotNeedlingMove 			REF= Service_Handshake.AllocationRobotNeedlingMove;
END_METHOD

METHOD PRIVATE ReferenceHMI
VAR_INPUT
END_VAR
Service_Handshake.AllocateMoveStructure REF= GVL_ADS.AllocateMoveStructure;
Service_Handshake.AllocateMoveStructure_Reverse REF= GVL_ADS.AllocateMoveStructure_Reverse;
Service_Handshake.EmptyRobotToTurnTableMove REF= GVL_ADS.EmptyRobotToTurnTableMove;
Service_Handshake.AllocateCircleMove REF= GVL_ADS.AllocateCircleMove;
Service_Handshake.TurnTableMove REF= GVL_ADS.TurnTableMove;
//Service_Handshake.AxesControl REF= GVL_ADS.AxesControl;
Service_Handshake.MachineReset REF= GVL_ADS.MachineReset;
Service_Handshake.RareFullBoxPush REF= GVL_ADS.RareFullBoxPush;
Service_Handshake.AutoMode_AllocateCircleMove REF= GVL_ADS.AutoMode_AllocateCircleMove;
Service_Handshake.AutoMode_RobotWarehouseMove REF= GVL_ADS.AutoMode_RobotWarehouseMove;
Service_Handshake.AutoMode_RobotAbsMove REF= GVL_ADS.AutoMode_RobotAbsMove;
Service_Handshake.AutoMode_EmptyBoxMove REF= GVL_ADS.AutoMode_EmptyBoxMove;
Service_Handshake.AutoMode_TurnTableMOve REF= GVL_ADS.AutoMode_TurnTableMOve;
Service_Handshake.AutoMode_AllocateMove REF= GVL_ADS.AutoMode_AllocateMove;
Service_Handshake.AutoMode_AllocateMove_Reverse REF= GVL_ADS.AutoMode_AllocateMove_Reverse;
Service_Handshake.AutoMode_AllocateBatchMode REF= GVL_ADS.AutoMode_AllocateBatchMode;
Service_Handshake.AutoMode_AllocateBatchMode_Reverse REF= GVL_ADS.AutoMode_AllocateBatchMode_Reverse;
Service_Handshake.AutoMode_SimpleAllocation_Batch REF= GVL_ADS.AutoMode_SimpleAllocation_Batch;
Service_Handshake.AutoMode_RareBoxMove REF= GVL_ADS.AutoMode_RareBoxMove;
Service_Handshake.AutoMode_OutBoxMove REF= GVL_ADS.AutoMode_OutBoxMove;
Service_Handshake.AutoMode_BoxMoveReverse REF= GVL_ADS.AutoMode_BoxMoveReverse;
Service_Handshake.AutoMode_WarehouseMove REF= GVL_ADS.AutoMode_WarehouseMove;
Service_Handshake.AutoMode_ErrorHandle REF= GVL_ADS.AutoMode_ErrorHandle;
Service_Handshake.AlarmAllocation REF= GVL_ADS.AlarmAllocation;
Service_Handshake.AutoMode_MoveConveyorJob REF= GVL_ADS.AutoMode_MoveConveyorJob;
Service_Handshake.AutoMode_WarehouseMotoWithRobotMove REF= GVL_ADS.AutoMode_WarehouseMotoWithRobotMove;
Service_Handshake.AutoMode_SimpleAllocate REF= GVL_ADS.AutoMode_SimpleAllocate;
Service_Handshake.AutoMode_PullOutConveyor REF= GVL_ADS.AutoMode_PullOutConveyor;
Service_Handshake.AutoMode_AddBoxes REF= GVL_ADS.AutoMode_AddBoxes;
Service_Handshake.MachineHome REF= GVL_ADS.MachineHome;
Service_Handshake.StorageRegionHome REF= GVL_ADS.StorageRegionHome;
Service_Handshake.AllocationRegionHome REF= GVL_ADS.AllocationRegionHome;
Service_Handshake.FGARegionHome REF= GVL_ADS.FGARegionHome;
Service_Handshake.StorageRegionMode REF= GVL_ADS.StorageRegionMode;
Service_Handshake.AllocationRegion REF= GVL_ADS.AllocationRegion;
Service_Handshake.FGARegionMode REF= GVL_ADS.FGARegionMode;
Service_Handshake.MachineMode REF= GVL_ADS.MachineMode;
Service_Handshake.OpPannel_Status REF= GVL_ADS.OpPannel_Status;
Service_Handshake.OpPannel_Ctrl REF= GVL_ADS.OpPannel_Ctrl;
Service_Handshake.FanucRobot_General REF= GVL_ADS.FanucRobot_General;
Service_Handshake.AutoMode_FeedInEmptyBoxWithRobot REF= GVL_ADS.AutoMode_FeedInEmptyBoxWithRobot;
Service_Handshake.AutoMode_ReloadRoundBeltBoxWithRobot REF= GVL_ADS.AutoMode_ReloadRoundBeltBoxWithRobot;
Service_Handshake.AutoMode_UpperFeedInConveyor REF= GVL_ADS.AutoMode_UpperFeedInConveyor;
//Service_Handshake.MachineState REF= GVL_ADS.MachineState;
Service_Handshake.AutoMode_RobotRegionMove_FeedInConveyor REF= GVL_ADS.AutoMode_RobotRegionMove_FeedInConveyor;
Service_Handshake.AutoMode_RobotRegionMove_AllocatedConveyor REF= GVL_ADS.AutoMode_RobotRegionMove_AllocatedConveyor;
Service_Handshake.AutoMode_RobotRegionMove_PullOutConveyor REF= GVL_ADS.AutoMode_RobotRegionMove_PullOutConveyor;
Service_Handshake.AutoMode_RobotRegionMove_BufferArea REF= GVL_ADS.AutoMode_RobotRegionMove_BufferArea;
Service_Handshake.AutoMode_RobotRegionMove_RoundBelt REF= GVL_ADS.AutoMode_RobotRegionMove_RoundBelt;
Service_Handshake.AutoMode_ShippingRobot_Left REF= GVL_ADS.AutoMode_ShippingRobot_Left;
Service_Handshake.AutoMode_ShippingRobot_Right REF= GVL_ADS.AutoMode_ShippingRobot_Right;
Service_Handshake.AutoMode_ShippingRobot_TransmitCVEnd REF= GVL_ADS.AutoMode_ShippingRobot_TransmitCVEnd;
Service_Handshake.AutoMode_SameSizeCVCamera REF= GVL_ADS.AutoMode_SameSizeCVCamera;
Service_Handshake.AutoMode_DifferentCVCamera REF= GVL_ADS.AutoMode_DifferentCVCamera;

Service_Handshake.AllocationRobotNeedlingMove REF= GVL_ADS.AllocationRobotNeedlingMove;
END_METHOD

METHOD RefShippingService
VAR_INPUT
END_VAR
ShippingService.AutoMode_ShippingRobot_Left REF= Service_Handshake.AutoMode_ShippingRobot_Left;
ShippingService.AutoMode_ShippingRobot_Right REF= Service_Handshake.AutoMode_ShippingRobot_Right;
ShippingService.AutoMode_ShippingRobot_TransmitCVEnd REF= Service_Handshake.AutoMode_ShippingRobot_TransmitCVEnd;
END_METHOD

METHOD PRIVATE RefStorageService
VAR_INPUT
END_VAR
StorageService.AutoMode_ReloadRoundBeltBoxWithRobot	REF= Service_Handshake.AutoMode_ReloadRoundBeltBoxWithRobot;
StorageService.AutoMode_FeedInEmptyBoxWithRobot REF= Service_Handshake.AutoMode_FeedInEmptyBoxWithRobot;
StorageService.AutoMode_RobotRegionMove_FeedInConveyor REF= Service_Handshake.AutoMode_RobotRegionMove_FeedInConveyor;
StorageService.AutoMode_RobotRegionMove_AllocatedConveyor REF= Service_Handshake.AutoMode_RobotRegionMove_AllocatedConveyor;
StorageService.AutoMode_RobotRegionMove_PullOutConveyor REF= Service_Handshake.AutoMode_RobotRegionMove_PullOutConveyor;
StorageService.AutoMode_RobotRegionMove_BufferArea REF= Service_Handshake.AutoMode_RobotRegionMove_BufferArea;
StorageService.AutoMode_RobotRegionMove_RoundBelt REF= Service_Handshake.AutoMode_RobotRegionMove_RoundBelt;
StorageService.AutoMode_UpperFeedInConveyor REF=  Service_Handshake.AutoMode_UpperFeedInConveyor;
StorageService.AutoMode_AddBoxes REF= Service_Handshake.AutoMode_AddBoxes;
StorageService.AutoMode_PullOutConveyor REF= Service_Handshake.AutoMode_PullOutConveyor;
StorageService.AutoMode_RobotAbsMove REF=  Service_Handshake.AutoMode_RobotAbsMove;
StorageService.AutoMode_WarehouseMotoWithRobotMove REF= Service_Handshake.AutoMode_WarehouseMotoWithRobotMove;
END_METHOD

END_FUNCTION_BLOCK

// ---- Library/00_PackML/01_ObjectBase/FB_ModeBase_V2.TcPOU
{attribute 'reflection'}
FUNCTION_BLOCK FB_ModeBase_V2 IMPLEMENTS I_UnitState, I_ErrorElement
VAR_INPUT
    eModeCommand  : E_UnitMode; // Mode from superior Unit
    eStateCommand : E_PMLCommand := ePMLCommand_Abort; // Command fro a new state from supterior unit
    PackTag       : REFERENCE TO ST_PackMLv30; // 
END_VAR
VAR_OUTPUT
    eModeCurrent  : E_UnitMode;
    eStateCurrent : E_PMLState;
END_VAR
VAR
    {attribute 'instance-path'}
    {attribute 'noinit'}
    _strName : STRING(255); // Instance path of the FB for Diagnostic

    fbUnitModeManager : PML_UnitModeManager; //The PML_UnitModeManager manage the Modechanges
    fbStateMachine    : PML_StateMachine; //The PML_StateMachine mangae the Statechanges

    eModeChange     : eModeChangeState; // This value is used to control mode change flow
    AllowModeChange : BOOL;
    nLastState      : E_PMLState; //Variable to store last state
    xError           : BOOL;
    xErrorID         : DINT;
    xErrorMsg        : T_MaxString;
	iErrorCount : INT;
	arAlarmTrigPtr : ARRAY[1..Tc3_PackML_V2.MaxAlarms] OF POINTER TO BOOL;
	arAlarmMsg : ARRAY[1..Tc3_PackML_V2.MaxAlarms] OF POINTER TO STRING;
	iErrorReflashIndex : INT;
END_VAR

CASE eModeChange OF
    eModeChangeState.WaitingRequest:
        // check unit is in the stand still, allow to change mode
        AllowModeChange := M_ModeChangeCheck();

        IF AllowModeChange AND (eModeCommand <> eModeCurrent) THEN
            eModeChange := eModeChangeState.StartingUnitModeManager;
        END_IF
    eModeChangeState.StartingUnitModeManager:
        fbUnitModeManager.bExecute             := TRUE;
        PackTag.Status.UnitModeChangeInProcess := TRUE;

        IF fbUnitModeManager.bDone THEN
            fbUnitModeManager.bExecute             := FALSE;
            eModeChange                            := eModeChangeState.WaitingRequest;
            PackTag.Status.UnitModeChangeInProcess := FALSE;
        ELSIF fbUnitModeManager.bError THEN
            fbUnitModeManager.bExecute := FALSE;
            nLastState                 := PackTag.Status.StateCurrent;
            eModeChange                := eModeChangeState.ErrorHandling;
        END_IF
    eModeChangeState.ErrorHandling:
        //ErrorHanddling
		eModeChange := 0; 
//        IF PackTag.Command.UnitModeChangeRequest THEN
//            eModeChange := 0;
//        ELSIF nLastState <> PackTag.Status.StateCurrent THEN
//            ;
//        END_IF
END_CASE

fbUnitModeManager(bExecute :=,
                  eModeCommand := eModeCommand,
                  eState := eStateCurrent,
                  eModeStatus => eModeCurrent,
                  sModeStatus =>,
                  bDone =>,
                  bError =>,
                  nErrorId =>);

IF fbUnitModeManager.eModeStatus <> E_UnitMode.Undefined THEN
    fbStateMachine(eMode := eModeCommand,
                   eCommand := eStateCommand,
                   stSubUnitInfoRef :=,
                   stOptions :=,
                   eState => eStateCurrent,
                   sState =>,
                   bError =>,
                   nErrorID =>);
END_IF

//One of the methods is executing  by the actual state
CASE eStateCurrent OF
    ePMLState_Undefined:
        M_Undefined();
    ePMLState_Clearing:
        M_Clearing();
    ePMLState_Stopped:
        M_Stopped();
    ePMLState_Starting:
        M_Starting();
    ePMLState_Idle:
        M_Idle();
    ePMLState_Suspended:
        M_Suspended();
    ePMLState_Execute:
        M_Execute();
    ePMLState_Stopping:
        M_Stopping();
    ePMLState_Aborting:
        M_Aborting();
    ePMLState_Aborted:
        M_Aborted();
    ePMLState_Holding:
        M_Holding();
    ePMLState_Held:
        M_Held();
    ePMLState_Unholding:
        M_Unholding();
    ePMLState_Suspending:
        M_Suspending();
    ePMLState_Unsuspending:
        M_Unsuspending();
    ePMLState_Resetting:
        M_Resetting();
    ePMLState_Completing:
        M_Completing();
    ePMLState_Complete:
        M_Complete();
END_CASE

Act_ErrorSync();

ACTION Act_ErrorSync:
FOR iErrorReflashIndex := 1 TO MaxAlarms DO
    IF arAlarmTrigPtr[iErrorReflashIndex] <> 0 THEN
        PackTag.Admin.Alarm[iErrorReflashIndex].Trigger := arAlarmTrigPtr[iErrorReflashIndex]^;
		//PackTag.Admin.Alarm[iErrorReflashIndex].Message := arAlarmMsg[iErrorReflashIndex]^;
    END_IF
END_FOR
END_ACTION

METHOD M_Aborted
M_StateComplete();
END_METHOD

METHOD M_Aborting
M_StateComplete();
END_METHOD

METHOD M_Clearing
M_StateComplete();
END_METHOD

METHOD M_Complete
M_StateComplete();
END_METHOD

METHOD M_Completing
M_StateComplete();
END_METHOD

METHOD M_Execute
M_StateComplete();
END_METHOD

METHOD M_GetError
VAR_INPUT
END_VAR
VAR_OUTPUT
	Error : BOOL;
	ErrorID : DINT;
	ErrorMsg : T_MaxString;
END_VAR
Error := xError;
ErrorID := xErrorID;
ErrorMsg := xErrorMsg;
END_METHOD

METHOD PUBLIC M_GetName :STRING
VAR_INPUT
END_VAR
M_GetName := _strName;
END_METHOD

METHOD M_Held
M_StateComplete();
END_METHOD

METHOD M_Holding
M_StateComplete();
END_METHOD

METHOD M_Idle
M_StateComplete();
END_METHOD

METHOD M_ModeChageAutoCheck : BOOL
VAR_INPUT
END_VAR
CASE eStateCurrent OF
	ePMLState_Aborted,ePMLState_Stopped,ePMLState_Idle :
		// Allow unit change mode to Auto
		M_ModeChageAutoCheck := TRUE;
	ePMLState_Undefined:
		M_ModeChageAutoCheck := TRUE;
END_CASE
END_METHOD

METHOD M_ModeChangeCheck : BOOL
VAR_INPUT
END_VAR
VAR_INST
    ManualAllowChange : BOOL;
    AutoAllowChange   : BOOL;
    HomingAllowChange : BOOL;
	MantainaceAllowChange : BOOL;
END_VAR
ManualAllowChange     := M_ModeChangeManualCheck();
AutoAllowChange       := M_ModeChageAutoCheck();
HomingAllowChange     := M_ModeChangeHomingCheck();
MantainaceAllowChange := M_ModeChangeMantainaceCheck();

M_ModeChangeCheck := ManualAllowChange AND AutoAllowChange AND HomingAllowChange AND MantainaceAllowChange;
END_METHOD

METHOD M_ModeChangeHomingCheck : BOOL
VAR_INPUT
END_VAR
CASE eStateCurrent OF
	ePMLState_Aborted,ePMLState_Stopped,ePMLState_Idle :
		// Allow unit change mode to Homing
		M_ModeChangeHomingCheck := TRUE;
	ePMLState_Undefined:
		M_ModeChangeHomingCheck := TRUE;

END_CASE
END_METHOD

METHOD M_ModeChangeMantainaceCheck : BOOL
VAR_INPUT
END_VAR
CASE eStateCurrent OF
	ePMLState_Aborted,ePMLState_Stopped,ePMLState_Idle :
		// Allow unit change mode to Mantainace
		M_ModeChangeMantainaceCheck := TRUE;
	ePMLState_Undefined:
		M_ModeChangeMantainaceCheck := TRUE;

END_CASE
END_METHOD

METHOD M_ModeChangeManualCheck : BOOL
VAR_INPUT
END_VAR
CASE eStateCurrent OF
	ePMLState_Aborted,ePMLState_Stopped,ePMLState_Idle :
		// Allow unit change mode to Manual
		M_ModeChangeManualCheck := TRUE;
	ePMLState_Undefined:
		M_ModeChangeManualCheck := TRUE;

END_CASE
END_METHOD

METHOD M_Resetting
M_StateComplete();
END_METHOD

METHOD M_Starting
M_StateComplete();
END_METHOD

METHOD M_StateComplete
//the actual state is completed
fbStateMachine.M_StateComplete();
END_METHOD

METHOD M_Stopped
M_StateComplete();
END_METHOD

METHOD M_Stopping
M_StateComplete();
END_METHOD

METHOD M_Suspended
M_StateComplete();
END_METHOD

METHOD M_Suspending
M_StateComplete();
END_METHOD

METHOD M_Undefined
M_StateComplete();
END_METHOD

METHOD M_Unholding
M_StateComplete();
END_METHOD

METHOD M_Unsuspending
M_StateComplete();
END_METHOD

METHOD RegisterAlarm
VAR_INPUT
    Trigger  : REFERENCE TO BOOL;
    ID       : DINT;
    value    : DINT;
    Message  : STRING;
    Category : DINT;
END_VAR
VAR_INST
    iLoopIndex : INT;
    HasSameID  : BOOL := FALSE;
    FoundIndex : INT := 0;
    FoundCount : INT := 0;
END_VAR
FOR iLoopIndex := 1 TO MaxAlarms DO
    IF PackTag.Admin.Alarm[iLoopIndex].ID = ID THEN
        IF NOT HasSameID THEN
            HasSameID := TRUE;
            FoundIndex := iLoopIndex;
			
			EXIT;
        END_IF
		PackTag.Admin.Alarm[iLoopIndex].Message := Message;
        FoundCount := FoundCount + 1;
    END_IF
END_FOR

IF NOT HasSameID THEN
    PackTag.Admin.Alarm[iErrorCount+1].ID := ID;
    PackTag.Admin.Alarm[iErrorCount+1].Value := value;
    PackTag.Admin.Alarm[iErrorCount+1].Message := Message;
    PackTag.Admin.Alarm[iErrorCount+1].Category := Category;
	arAlarmTrigPtr[iErrorCount+1] := ADR(Trigger);
	//arAlarmMsg[iErrorCount+1] := ADR(Message);
	iErrorCount := iErrorCount +1 ;
END_IF
END_METHOD

END_FUNCTION_BLOCK

// ---- Library/10_Machine/18_HMI_Handshake/FB_HmiHandShake.TcPOU
FUNCTION_BLOCK FB_HmiHandShake EXTENDS BATW_Base.FB_ActionBasic
VAR_INPUT
    xEnable        : BOOL;
    CylinderStatus : ST_CylinderStatus;
    MotorStatus    : ST_MotorStatus;
    AxesStatus     : ST_AXES_STATUS;
	FanucRobot : REFERENCE TO UNI_FanucRobotList;
END_VAR
VAR_OUTPUT
	//AllocatingManual : st_ads_AllocateMoveStructure;
END_VAR
VAR
    StateBehaviour : CBML.LConC;
	//HMI_Handshake_Old : REFERENCE TO ST_HMI_Handshake;
END_VAR

THIS^.IBehaviourModel := StateBehaviour;
StateBehaviour(xEnable := xEnable, xBusy => xBusy, xError => xError);

METHOD CleanupAction
VAR_INPUT
    xAbortProposed   : BOOL;
    iErrorIDProposed : INT;
END_VAR
VAR_OUTPUT
    xComplete : BOOL := TRUE;
    xAbort    : BOOL := xAbortProposed;
    iErrorID  : INT := iErrorIDProposed;
END_VAR
END_METHOD

METHOD CyclicAction
VAR_INPUT
    itfTimingController : CBML.ITimingController;
END_VAR
VAR_OUTPUT
    xComplete : BOOL := TRUE;
    iErrorID  : INT := 0;
END_VAR
GetIOStatus();
GetAxesStatus();
GetMotorStatus();
GetCylinderStatus();
SetMachineParemeter();
//AllocatingManual := GVL_ADS.AllocateMoveStructure;
FanucRobot.List.StorageRobot.VelocityCommand := LREAL_TO_INT( GVL_HMI.Setup.StorageRobot.RobotVelocity);
FanucRobot.List.ShippingRobot.VelocityCommand := LREAL_TO_INT( GVL_HMI.Setup.ShippingRobot.RobotVelocity);
END_METHOD

METHOD ExitAction
VAR_INPUT
    xAfterCleanup : BOOL;
    xInCopyCode   : BOOL;
END_VAR
END_METHOD

(* This method is used to read DAS servo status and send to GVL_HMI
*)
METHOD PRIVATE GetAxesStatus
VAR_INPUT
END_VAR
// Read Axes status
GVL_HMI.Status.Axes.Allocate_X := M_GetAxisStatus(AxisNo.Allocate_X);
GVL_HMI.Status.Axes.Allocate_Y := M_GetAxisStatus(AxisNo.Allocate_Y);
GVL_HMI.Status.Axes.OutRobot_X := M_GetAxisStatus(AxisNo.OutRobot_X);
GVL_HMI.Status.Axes.OutRobot_Y := M_GetAxisStatus(AxisNo.OutRobot_Y);
GVL_HMI.Status.Axes.RoundBelt := M_GetAxisStatus(AxisNo.RoundBelt);
GVL_HMI.Status.Axes.TurnTable := M_GetAxisStatus(AxisNo.TurnTable);
GVL_HMI.Status.Axes.RackMotor := M_GetAxisStatus(AxisNo.RackMotor);
END_METHOD

METHOD PRIVATE GetCylinderStatus
VAR_INPUT
END_VAR
GVL_HMI.Status.Cylinders := CylinderStatus;
END_METHOD

METHOD PRIVATE GetIOStatus
VAR_INPUT
END_VAR
// Read  PLC Input Signal
GVL_HMI.IOMonitor.Input.X0  := GVL_Input.uniDI.stDIList.X0;
GVL_HMI.IOMonitor.Input.X1  := GVL_Input.uniDI.stDIList.X1;
GVL_HMI.IOMonitor.Input.X2  := GVL_Input.uniDI.stDIList.X2;
GVL_HMI.IOMonitor.Input.X3  := GVL_Input.uniDI.stDIList.X3;
GVL_HMI.IOMonitor.Input.X4  := GVL_Input.uniDI.stDIList.X4;
//GVL_HMI.IOMonitor.Input.X5  := GVL_Input.uniDI.stDIList.X0;
GVL_HMI.IOMonitor.Input.X6  := GVL_Input.uniDI.stDIList.X6;
GVL_HMI.IOMonitor.Input.X7  := GVL_Input.uniDI.stDIList.X7;
GVL_HMI.IOMonitor.Input.X8  := GVL_Input.uniDI.stDIList.X8;
GVL_HMI.IOMonitor.Input.X9  := GVL_Input.uniDI.stDIList.X9;
GVL_HMI.IOMonitor.Input.X10  := GVL_Input.uniDI.stDIList.X10;
GVL_HMI.IOMonitor.Input.X11  := GVL_Input.uniDI.stDIList.X11;
// Read PLC Output signal
GVL_HMI.IOMonitor.Output := GVL_Output.uniDO.stDIList;
// Read Wheelhous ModbusRTU sensor signal
GVL_HMI.IOMonitor.Input.arWheelhouseInput := ComModbusRTU.arr485sensor;
END_METHOD

METHOD PRIVATE GetMotorStatus
VAR_INPUT
END_VAR
GVL_HMI.Status.Motor := MotorStatus;
END_METHOD

(* This method is used to read single axis status accroding AxisNo
*)
METHOD M_GetAxisStatus : ST_SINGLEAXIS_STATUS
VAR_INPUT
	AxisNo : AxisNo;
END_VAR
M_GetAxisStatus.ActPos := arAxisCtrl_gb[AxisNo].Admin.Axis.NcToPlc.ActPos;
M_GetAxisStatus.ActVel := arAxisCtrl_gb[AxisNo].Admin.Axis.NcToPlc.ActVelo;
M_GetAxisStatus.Error := arAxisCtrl_gb[AxisNo].Admin.Axis.Status.Error;
IF AxisNo = 4 THEN
	M_GetAxisStatus.Homed := GVL_Machine.AllocatYAxisHome;
ELSE
	M_GetAxisStatus.Homed := arAxisCtrl_gb[AxisNo].Admin.Axis.Status.Homed;
END_IF

M_GetAxisStatus.CmdDone := arAxisStatus_gb[AxisNo].Admin.CmdDone;
M_GetAxisStatus.DriveTemp := 400;
M_GetAxisStatus.MotorTemp := 600;
END_METHOD

METHOD ResetAction
VAR_OUTPUT
    xComplete : BOOL := TRUE;
END_VAR
END_METHOD

METHOD PRIVATE SetMachineParemeter
VAR_INPUT
END_VAR
GVL_Machine.RemoteData := GVL_HMI.Setup;
END_METHOD

METHOD StartAction
VAR_OUTPUT
    xComplete : BOOL := TRUE;
    iErrorID  : INT := 0;
END_VAR
END_METHOD

END_FUNCTION_BLOCK

// ---- Library/20_MachineUnits/22_AllocateArea/FB_AllocateAreaWithRoundbelt.TcPOU
FUNCTION_BLOCK FB_AllocateAreaWithRoundbelt EXTENDS FB_ModeBase_V2 IMPLEMENTS I_UnitState
VAR_INPUT
    INPUT       : REFERENCE TO ST_InputTable;
    OUTPUT      : REFERENCE TO ST_OutputTable;
    CurrentData : ST_SetupPara;
    // Componets
    Cylinder : REFERENCE TO UNI_CylinderList;
    Service  : REFERENCE TO ST_AllocateService;
    Motor    : REFERENCE TO UNI_MotorList;
    Reset            : REFERENCE TO BOOL;
	Stop :  REFERENCE TO BOOL;
	bStopMem : REFERENCE to BOOL;
END_VAR
VAR_OUTPUT
	Homed : BOOL;
END_VAR
VAR
    InitDone          : BOOL;
    Clip              : U_Cylinders;
    Cylinders         : U_Cylinders;
    OutRobotCylinders : Uni_DuoCylinders;
    OutRobotClips     : Uni_DuoCylinders;

    i : INT;
    //============== Service====================
    // Allocate Home
    fbAllocateHome : FB_AllocateAreaHome;
    //RoundBelt
    RoundBeltControl  : FB_RoundBeltService;
    _RoundBeltMoveJob : st_AllocateCircleMoveStructure;
    //RoundBeltMoveJob_Internal 	: st_AllocateCircleMoveStructure;		
    RoundBeltControlAccess               : E_RoundBeltControlAccess := E_RoundBeltControlAccess.Host;
    RoundBeltMoveJob_Ctrl                : ST_CommandBasic;
    RoundBeltMoveJob_Ctrl_Batch          : ST_CommandBasic;
    RoundBeltMoveJob_Status              : ST_StatusBasic;
    RoundBeltMoveJob_Position            : LREAL;
    RoundBeltMoveJob_Position_FanucRobot : LREAL;
    //TurnTable
    TurnTableControl : FB_TurnTableService;

    //Allocating
    fb_AllocateBatchMode        : FB_AllocateMoveAutoBatchMode;
    AutoAllocateJobBatch_Ctrl   : st_AllocateMoveAutoBatchMode_Ctrl;
    AutoAllocateJobBatch_Status : st_AllocateMoveAutoBatchMode_Status;
    bAutoAllocateJobDryRun      : BOOL;

	  //Allocating reverse
    fb_AllocateBatchMode_Reverse        : FB_AllocateMoveAutoBatchMode_Reverse;
    AutoAllocateJobBatch_Reverse_Ctrl   : st_AllocateMoveAutoBatchMode_Ctrl;
    AutoAllocateJobBatch_Reverse_Status : st_AllocateMoveAutoBatchMode_Status;
   
	
    //OutRobot EmptyBoxMove
    fbOutRobot_EmptyBoxMove        : FB_OutRobot_EmptyBoxMove;
    fbOutRobot_EmptyBoxMove_Ctrl   : ST_CommandBasic;
    fbOutRobot_EmptyBoxMove_Status : ST_StatusBasic;

    //OutRobot RareBoxMove
    fbOutRobot_RareBoxMove        : FB_OutRobot_RareBoxMove;
    fbOutRobot_RareBoxMove_Ctrl   : ST_CommandBasic;
    fbOutRobot_RareBoxMove_Status : ST_StatusBasic;

    //OutRobot BoxMoveReverse	
    fbOutRobot_BoxMoveReverse        : FB_OutRobot_BoxMoveReverse;
    fbOutRobot_BoxMoveReverse_Ctrl   : ST_CommandBasic;
    fbOutRobot_BoxMoveReverse_Status : ST_StatusBasic;

	//OutRobot TurnTable to RoundBelt
	fbOutRobot_TurnTableToRoundBelt: FB_OutRobot_BoxMoveTurnTableToRoundBelt;
	fbOutRobot_TurnTableToRoundBel_Ctrl   : ST_CommandBasic;
    fbOutRobot_TurnTableToRoundBel_Status : ST_StatusBasic;
	
    //TransCV Camera
    fbSameSizeCVCamera  : FB_SameSizeCVCamera;
    fbDifferentCVCamera : FB_DifferentCVCamera;
	TransCV_Press 		: BOOL :=FALSE;

    // Round belt
    AutoRotatebelt_Internal_Ctrl   : st_RoundBeltAutoSingleMove_Ctrl;
    AutoRotatebelt_Internal_Status : st_RoundBeltAutoSingleMove_Status;
    _AutoRotatebelt_Ctrl           : st_RoundBeltAutoSingleMove_Ctrl;
    _AutoRotatebelt_Status         : st_RoundBeltAutoSingleMove_Status;
    bInternalRotateBeltRequest     : BOOL;
    bReloadRotateBeltRequest       : BOOL;

    // Pullout

    fbPulloutCV                 : FB_PullOutConveyorAction;
    _AutoPullout_Ctrl           : ST_AutoPullOutConveyorCommand;
    _AutoPullout_Status         : ST_AutoPullOutConveyorSatus;
    _AutoPullout_Info           : ST_PullOutConveyorInfo;
    AutoPullout_Internal_Ctrl   : ST_AutoPullOutConveyorCommand;
    AutoPullout_Internal_Status : ST_AutoPullOutConveyorSatus;
    AutoPullout_Internal_Info   : ST_PullOutConveyorInfo;
    RobotPullout_Internal_Ctrl   : ST_AutoPullOutConveyorCommand;
    RobotPullout_Internal_Status : ST_AutoPullOutConveyorSatus;
    RobotPullout_Internal_Info   : ST_PullOutConveyorInfo;
	fbPulloutCV_BTNCtrl			:FB_PullOutConveyorBtnCtrl;

    PulloutControlAccess        : E_RoundBeltControlAccess := E_RoundBeltControlAccess.Host;
    bPulloutConveyorInternCtrl  : BOOL;
	
	// TurnTable
	 _TurnTableMove                      :  st_ads_OneAxisMoveWithPosition;
	 
	 //AllocateRobotNeedlingMove
	 fbAllocateRobotNeedlingMove		: FB_AllocateRobotNeedlingMove;

END_VAR

SUPER^();
IF __ISVALIDREF(PackTag)  THEN
	
    eModeCommand  := PackTag.Command.UnitMode;
    eStateCommand := PackTag.Command.CntrlCmd;
ELSE
    RETURN;
END_IF

IF __ISVALIDREF(Cylinder) THEN
	
	Clip.stCylinders.Cylinder0 REF= Cylinder.List.fbAllocateRobot_LeftClamp1;
	Clip.stCylinders.Cylinder1 REF= Cylinder.List.fbAllocateRobot_LeftClamp2;
	Clip.stCylinders.Cylinder2 REF= Cylinder.List.fbAllocateRobot_RightClamp1;
	Clip.stCylinders.Cylinder3 REF= Cylinder.List.fbAllocateRobot_RightClamp2;
	Cylinders.stCylinders.Cylinder0 REF= Cylinder.List.fbAllocateRobot_LeftVert1;
	Cylinders.stCylinders.Cylinder1 REF= Cylinder.List.fbAllocateRobot_LeftVert2;
	Cylinders.stCylinders.Cylinder2 REF= Cylinder.List.fbAllocateRobot_RightVert1;
	Cylinders.stCylinders.Cylinder3 REF= Cylinder.List.fbAllocateRobot_RightVert2;
	
	OutRobotCylinders.stCylinders.Cylinder1 REF= Cylinder.List.fbOutRobot_AsideVert;
	OutRobotCylinders.stCylinders.Cylinder2 REF= Cylinder.List.fbOutRobot_BsideVert;
	OutRobotClips.stCylinders.Cylinder1 REF= Cylinder.List.fbOutRobot_AsideClamp;
	OutRobotClips.stCylinders.Cylinder2 REF= Cylinder.List.fbOutRobot_BsideClamp;
	
END_IF

ACTION A00_Service:
fbAllocateHome(
	xDone=> , 
	xBusy=> , 
	xError=> , 
	xExecute:= , 
	xAbort:= ,
	Homed := Homed, 
	Cylinder:= Cylinder, 
	Motor:= Motor, 
	CurrentData:= CurrentData, 
	TimeOut:= , 
	xAborted=> , 
	iErrorID=> , 
	ErrorMsg=> ,
	AxisHomingRequest =>);
	//Service.AllocateRegionHome.Homed:= bHomed;

RoundBeltControl(
	xDone=> _RoundBeltMoveJob.HandShake.Done, 
	xBusy=> _RoundBeltMoveJob.HandShake.Busy, 
	xError=> _RoundBeltMoveJob.HandShake.Error, 
	xExecute:= _RoundBeltMoveJob.HandShake.Execute, 
	xAbort:= , 
	TargetStation:= LREAL_TO_INT( _RoundBeltMoveJob.Position), 
	Cylinder:= Cylinder, 
	TimeOut:= , 
	xAborted=> , 
	iErrorID=> , 
	ErrorMsg=> );
	
TurnTableControl(
	xDone=> _TurnTableMove.HandShake.Done, 
	xBusy=> _TurnTableMove.HandShake.Busy, 
	xError=> _TurnTableMove.HandShake.Error, 
	xExecute:= _TurnTableMove.HandShake.Execute, 
	xAbort:= , 
	iTurnTableTarget:= LREAL_TO_INT(_TurnTableMove.Position), 
	Cylinder:= Cylinder, 
	TimeOut:= , 
	xAborted=> , 
	iErrorID=> , 
	ErrorMsg=> );
	
fb_AllocateBatchMode(
	Execute:= AutoAllocateJobBatch_Ctrl.bExecute, 
	Abort:= , 
	Reset:= Reset, 
	ObjectName:= 'Allocate One process', 
	Busy=> AutoAllocateJobBatch_Status.bBusy, 
	Done=> AutoAllocateJobBatch_Status.bDone, 
	Aborted=> , 
	Error=> AutoAllocateJobBatch_Status.bError, 
	ErrorID=>AutoAllocateJobBatch_Status.ErrorID , 
	Status=>AutoAllocateJobBatch_Status.Status , 
	UniqueErrorCode=> , 
	Pause:=bStopMem , 
	SimpleAllocateMode:= AutoAllocateJobBatch_Ctrl.bSimpleAllocation, 
	bOccupied:=AutoAllocateJobBatch_Ctrl.bOccupied, 
	Clips:= Clip.Cylinders, 
	cylinders:= Cylinders.Cylinders, 
	TurnTable_Press:= Cylinder.List.fbTurntable_Press, 
	RoundBelt_Press:= Cylinder.List.fbRoundBelt_WorkZone_Press, 
	AutoAllocateJobBatch_Ctrl:= AutoAllocateJobBatch_Ctrl, 
	INPUT:= INPUT, 
	OUTPUT:= OUTPUT, 
	NrOfAllocateCylinder:= 4, 
	CurrentData:= CurrentData, 
	bAutoAllocateJobDryRun:= bAutoAllocateJobDryRun, // Dry run : No round belt move
	ProcessedIndex=> AutoAllocateJobBatch_Status.iIndex,
	RoundBeltMoveJob_Ctrl =>,
	RoundBeltMoveJob_Status := RoundBeltMoveJob_Status,
	RoundBeltMoveJob_Position =>	 );
	
	IF fb_AllocateBatchMode.SimpleAllocateMode THEN
		 Service.AutoMode_SimpleAllocation_Batch.WorkedID:= AutoAllocateJobBatch_Status.iIndex;
	ELSE
		 Service.AutoMode_AllocateBatchMode.WorkedID:= AutoAllocateJobBatch_Status.iIndex;
	END_IF
fb_AllocateBatchMode_Reverse(
	Execute:=AutoAllocateJobBatch_Reverse_Ctrl.bExecute , 
	Abort:= , 
	Reset:= Reset, 
	ObjectName:= 'Allocate batch reverse', 
	Busy=> AutoAllocateJobBatch_Reverse_Status.bBusy, 
	Done=> AutoAllocateJobBatch_Reverse_Status.bDone, 
	Aborted=> AutoAllocateJobBatch_Reverse_Status.bAborted, 
	Error=> AutoAllocateJobBatch_Reverse_Status.bError, 
	ErrorID=> AutoAllocateJobBatch_Reverse_Status.ErrorID, 
	Status=> AutoAllocateJobBatch_Reverse_Status.Status, 
	UniqueErrorCode=> , 
	Pause:= bStopMem,  
	bOccupied:= AutoAllocateJobBatch_Reverse_Ctrl.bOccupied, 
	Clips:= Clip.Cylinders, 
	cylinders:= Cylinders.Cylinders, 
	TurnTable_Press:= Cylinder.List.fbTurntable_Press, 
	RoundBelt_Press:= Cylinder.List.fbRoundBelt_WorkZone_Press, 
	AutoAllocateJobBatch_Reverse_Ctrl:= AutoAllocateJobBatch_Reverse_Ctrl, 
	INPUT:= INPUT, 
	OUTPUT:= OUTPUT, 
	NrOfAllocateCylinder:=4 , 
	CurrentData:= CurrentData, 
	bAutoAllocateJobDryRun:= bAutoAllocateJobDryRun, 
	RoundBeltMoveJob_Ctrl=> , 
	ProcessedIndex=> AutoAllocateJobBatch_Reverse_Status.iIndex,
	RoundBeltMoveJob_Status := RoundBeltMoveJob_Status,
	RoundBeltMoveJob_Position =>);

	
fbOutRobot_EmptyBoxMove(
	Execute:= Service.AutoMode_EmptyBoxMove.HandShake.Execute, 
	Abort:= , 
	Reset:= Reset , 
	ObjectName:= 'fbOutRobot_EmptyBoxMove', 
	Busy=> Service.AutoMode_EmptyBoxMove.HandShake.Busy, 
	Done=> Service.AutoMode_EmptyBoxMove.HandShake.Done, 
	Aborted=> , 
	Error=> Service.AutoMode_EmptyBoxMove.HandShake.Error, 
	ErrorID=> , 
	Status=> , 
	UniqueErrorCode=> , 
	INPUT:= INPUT, 
	Cylinder:= Cylinder, 
	Motor:= Motor, 
	Cylinders :=OutRobotCylinders.Cylinders,
	Clips := OutRobotClips.Cylinders,
	AutoMode_OutRobotMoveMove:=Service.AutoMode_EmptyBoxMove );

fbOutRobot_RareBoxMove(
	Execute:= Service.AutoMode_RareBoxMove.HandShake.Execute , 
	Abort:= , 
	Reset:= Reset, 
	ObjectName:= 'fbOutRobot_RareBoxMove', 
	Busy=> Service.AutoMode_RareBoxMove.HandShake.Busy, 
	Done=> Service.AutoMode_RareBoxMove.HandShake.Done, 
	Aborted=> , 
	Error=> Service.AutoMode_RareBoxMove.HandShake.Error, 
	ErrorID=> , 
	Status=> , 
	UniqueErrorCode=> , 
	INPUT:=INPUT , 
	Cylinder:= Cylinder, 
	Motor:= Motor, 
	Cylinders :=OutRobotCylinders.Cylinders,
	Clips := OutRobotClips.Cylinders,
	AutoMode_OutRobotMoveMove:= Service.AutoMode_RareBoxMove);

fbOutRobot_BoxMoveReverse(
	Execute:= Service.AutoMode_BoxMoveReverse.HandShake.Execute, 
	Abort:= , 
	Reset:= Reset, 
	ObjectName:='fbOutRobot_BoxMoveReverse', 
	Busy=> Service.AutoMode_BoxMoveReverse.HandShake.Busy, 
	Done=> Service.AutoMode_BoxMoveReverse.HandShake.Done, 
	Aborted=> , 
	Error=> Service.AutoMode_BoxMoveReverse.HandShake.Error, 
	ErrorID=> , 
	Status=> , 
	UniqueErrorCode=> , 
	INPUT:= INPUT, 
	Cylinder:= Cylinder, 
	Motor:= Motor, 
	Cylinders :=OutRobotCylinders.Cylinders,
	Clips := OutRobotClips.Cylinders,
	AutoMode_OutRobotMoveMove:= Service.AutoMode_BoxMoveReverse);	
	
fbDifferentCVCamera(
	xDone=> Service.AutoMode_DifferentCVCamera.Status.Done, 
	xBusy=> Service.AutoMode_DifferentCVCamera.Status.Busy, 
	xError=> Service.AutoMode_DifferentCVCamera.Status.Error, 
	xExecute:= Service.AutoMode_DifferentCVCamera.Command.Execute, 
	xAbort:= Service.AutoMode_DifferentCVCamera.Command.Abort, 
	xReset:= Reset, 
	Cylinder:= Cylinder, 
	TimeOut:= , 
	Input:= INPUT, 
	OutPut:= OutPut ,
	Motor:= Motor, 
	BoxCameraDone:= Service.AutoMode_DifferentCVCamera.BoxCameraDone, 
	xAborted=> , 
	iErrorID=> , 
	ErrorMsg=> , 
	UseBoxCamera=> Service.AutoMode_DifferentCVCamera.UseBoxCamera);

fbOutRobot_TurnTableToRoundBelt(
	Execute:= fbOutRobot_TurnTableToRoundBel_Ctrl.Execute, 
	Abort:= fbOutRobot_TurnTableToRoundBel_Ctrl.Abort, 
	Reset:= Reset, 
	ObjectName:= 'fbOutRobot_TurnTableToRoundBelt', 
	Busy=> fbOutRobot_TurnTableToRoundBel_Status.Busy, 
	Done=> fbOutRobot_TurnTableToRoundBel_Status.Done, 
	Aborted=> , 
	Error=> fbOutRobot_TurnTableToRoundBel_Status.Error, 
	ErrorID=> , 
	Status=> fbOutRobot_TurnTableToRoundBel_Status.Status, 
	UniqueErrorCode=> , 
	INPUT:= INPUT, 
	Cylinders:= OutRobotCylinders.Cylinders, 
	Clips:=OutRobotClips.Cylinders , 
	AutoMode_TurnTableToRoundBelt:= ); // todo creative var to fill in cmooand info	
	
	fbSameSizeCVCamera(
		xReset := Reset,
		xDone=> Service.AutoMode_SameSizeCVCamera.Status.Done, 
		xBusy=> Service.AutoMode_SameSizeCVCamera.Status.Busy, 
		xError=> Service.AutoMode_SameSizeCVCamera.Status.Error, 
		xExecute:= Service.AutoMode_SameSizeCVCamera.Command.Execute, 
		xAbort:= Service.AutoMode_SameSizeCVCamera.Command.Abort, 
		Cylinder:= Cylinder, 
		TimeOut:= , 
		Input:= INPUT, 
		OutPut:= OUTPUT, 
		Motor:= Motor, 
		BoxCameraDone:= Service.AutoMode_SameSizeCVCamera.BoxCameraDone, 
		xAborted=> , 
		iErrorID=> , 
		ErrorMsg=> , 
		UseBoxCamera=> Service.AutoMode_SameSizeCVCamera.UseBoxCamera);
	
	
	
fbPulloutCV(
	Execute:= _AutoPullout_Ctrl.Execute, 
	Abort:= _AutoPullout_Ctrl.Abort, 
	Reset:= Reset, 
	ObjectName:= ' Pullout conveyor ', 
	Busy=> _AutoPullout_Status.Busy, 
	Done=> _AutoPullout_Status.Done, 
	Aborted=> , 
	Error=> _AutoPullout_Status.Error, 
	ErrorID=> , 
	Status=> _AutoPullout_Status.Status, 
	UniqueErrorCode=> , 
	FixCylinderA1:= Cylinder.List.fbPullOutCV_AsidePress1, 
	FixCylinderA2:= Cylinder.List.fbPullOutCV_AsidePress2, 
	FixCylinderB1:= Cylinder.List.fbPullOutCV_BsidePress1, 
	FixCylinderB2:= Cylinder.List.fbPullOutCV_BsidePress2, 
	BarrierCylinderA:= Cylinder.List.fbPullOutCV_AsideBlock, 
	BarrierCylinderB:= Cylinder.List.fbPullOutCV_BsideBlock, 
	ConveyorMotorA:= Motor.List.PullOutCV_A, 
	ConveyorMotorB:= Motor.List.PullOutCV_B, 
	INPUT:= INPUT, 
	PullOutInfo:= _AutoPullout_Info);
	
fbPulloutCV_BTNCtrl(
	Input:= INPUT, 
	Output:= OUTPUT, 
	Motor:= Motor, 
	bPullOutConveyorExecute:= _AutoPullout_Ctrl.Execute, 
	bPullOutConveyorDone:= _AutoPullout_Status.Done, 
	bPullOutConveyorBusy:= _AutoPullout_Status.Busy, 
	StroageRegionMode:= eModeCurrent, 
	PullOutConveyorState=> );
	
fbAllocateRobotNeedlingMove(
	xDone=>  Service.AllocateRobotNeedlingMove.Status.Done,
	xBusy=> Service.AllocateRobotNeedlingMove.Status.Busy, 
	xError=> Service.AllocateRobotNeedlingMove.Status.Error, 
	xExecute:= Service.AllocateRobotNeedlingMove.Command.Execute, 
	xAbort:= Service.AllocateRobotNeedlingMove.Command.Abort, 
	TimeOut:= , 
	MovingInfo:= Service.AllocateRobotNeedlingMove.MovingInfo, 
	xAborted=> , 
	iErrorID=> , 
	ErrorMsg=> Service.AllocateRobotNeedlingMove.Status.Status);
END_ACTION

ACTION A01_RoundBeltAccessControl:
CASE RoundBeltControlAccess OF 
	E_RoundBeltControlAccess.Host :
	 IF eModeCurrent = E_UnitMode.Manual THEN
		_RoundBeltMoveJob.Position :=Service.AllocateCircleMove.Position;
		_RoundBeltMoveJob.Latch :=Service.AllocateCircleMove.Latch;
		_RoundBeltMoveJob.HandShake.Execute :=Service.AllocateCircleMove.HandShake.Execute;
		_RoundBeltMoveJob.HandShake.Reset :=Service.AllocateCircleMove.HandShake.Reset;
		_RoundBeltMoveJob.HandShake.Occupied  :=Service.AllocateCircleMove.HandShake.Occupied;
		Service.AllocateCircleMove.HandShake.Busy := _RoundBeltMoveJob.HandShake.Busy;
		Service.AllocateCircleMove.HandShake.Done := _RoundBeltMoveJob.HandShake.Done;
		Service.AllocateCircleMove.HandShake.Error := _RoundBeltMoveJob.HandShake.Error;
	ELSIF  eModeCurrent = E_UnitMode.Auto THEN
		_RoundBeltMoveJob.Position :=Service.AutoMode_AllocateCircleMove.Position;
		_RoundBeltMoveJob.Latch :=Service.AutoMode_AllocateCircleMove.Latch;
		_RoundBeltMoveJob.HandShake.Execute :=Service.AutoMode_AllocateCircleMove.HandShake.Execute;
		_RoundBeltMoveJob.HandShake.Reset :=Service.AutoMode_AllocateCircleMove.HandShake.Reset;
		_RoundBeltMoveJob.HandShake.Occupied  :=Service.AutoMode_AllocateCircleMove.HandShake.Occupied;
		Service.AutoMode_AllocateCircleMove.HandShake.Busy := _RoundBeltMoveJob.HandShake.Busy;
		Service.AutoMode_AllocateCircleMove.HandShake.Done := _RoundBeltMoveJob.HandShake.Done;
		Service.AutoMode_AllocateCircleMove.HandShake.Error := _RoundBeltMoveJob.HandShake.Error;
	END_IF
		
	E_RoundBeltControlAccess.Allocating  :
	
		_RoundBeltMoveJob.Position :=RoundBeltMoveJob_Position;
		//_RoundBeltMoveJob.Latch :=;
		_RoundBeltMoveJob.HandShake.Execute :=RoundBeltMoveJob_Ctrl_Batch.Execute;
		_RoundBeltMoveJob.HandShake.Reset :=RoundBeltMoveJob_Ctrl_Batch.Reset;
		RoundBeltMoveJob_Status.Busy := _RoundBeltMoveJob.HandShake.Busy;
		RoundBeltMoveJob_Status.Done := _RoundBeltMoveJob.HandShake.Done;
		RoundBeltMoveJob_Status.Error := _RoundBeltMoveJob.HandShake.Error;

	E_RoundBeltControlAccess.FanucRobot:
		_RoundBeltMoveJob.Position :=RoundBeltMoveJob_Position_FanucRobot;
		//_RoundBeltMoveJob.Latch :=;
		_RoundBeltMoveJob.HandShake.Execute :=RoundBeltMoveJob_Ctrl.Execute;
		_RoundBeltMoveJob.HandShake.Reset :=RoundBeltMoveJob_Ctrl.Reset;
		RoundBeltMoveJob_Status.Busy := _RoundBeltMoveJob.HandShake.Busy;
		RoundBeltMoveJob_Status.Done := _RoundBeltMoveJob.HandShake.Done;
		RoundBeltMoveJob_Status.Error := _RoundBeltMoveJob.HandShake.Error;	
END_CASE
END_ACTION

ACTION A02_PulloutAccessControl:
CASE PulloutControlAccess OF
    E_RoundBeltControlAccess.Host:
        _AutoPullout_Ctrl.Execute := Service.AutoMode_PullOutConveyor.Command.Execute;
        _AutoPullout_Ctrl.Abort := Service.AutoMode_PullOutConveyor.Command.Abort;
        _AutoPullout_Ctrl.Reset := Service.AutoMode_PullOutConveyor.Command.Reset;
        Service.AutoMode_PullOutConveyor.Status.Busy := _AutoPullout_Status.Busy;
        Service.AutoMode_PullOutConveyor.Status.Done := _AutoPullout_Status.Done;
        Service.AutoMode_PullOutConveyor.Status.Error := _AutoPullout_Status.Error;
        Service.AutoMode_PullOutConveyor.Status.Status := _AutoPullout_Status.Status;
        _AutoPullout_Info := Service.AutoMode_PullOutConveyor.PullOutConveyorInfo;
    E_RoundBeltControlAccess.Allocating:
        _AutoPullout_Ctrl.Execute := AutoPullout_Internal_Ctrl.Execute;
        _AutoPullout_Ctrl.Abort := AutoPullout_Internal_Ctrl.Abort;
        _AutoPullout_Ctrl.Reset := AutoPullout_Internal_Ctrl.Reset;
        AutoPullout_Internal_Status.Busy := _AutoPullout_Status.Busy;
        AutoPullout_Internal_Status.Done := _AutoPullout_Status.Done;
        AutoPullout_Internal_Status.Error := _AutoPullout_Status.Error;
        AutoPullout_Internal_Status.Status := _AutoPullout_Status.Status;
        _AutoPullout_Info := AutoPullout_Internal_Info;
    E_RoundBeltControlAccess.FanucRobot:
        _AutoPullout_Ctrl.Execute := RobotPullout_Internal_Ctrl.Execute;
        _AutoPullout_Ctrl.Abort := RobotPullout_Internal_Ctrl.Abort;
        _AutoPullout_Ctrl.Reset := RobotPullout_Internal_Ctrl.Reset;
        RobotPullout_Internal_Status.Busy := _AutoPullout_Status.Busy;
        RobotPullout_Internal_Status.Done := _AutoPullout_Status.Done;
        RobotPullout_Internal_Status.Error := _AutoPullout_Status.Error;
        RobotPullout_Internal_Status.Status := _AutoPullout_Status.Status;
        _AutoPullout_Info := RobotPullout_Internal_Info;
END_CASE
END_ACTION

ACTION A99_ErrorHandler:

END_ACTION

METHOD M_Aborted
M_StateComplete();
END_METHOD

METHOD M_Aborting
M_StateComplete();
END_METHOD

METHOD M_ActiveRoundBeltInternalCtrl : BOOL
VAR_INPUT
END_VAR
bReloadRotateBeltRequest := TRUE;
M_ActiveRoundBeltInternalCtrl := true; // Method end
END_METHOD

METHOD PRIVATE M_AutoAllocatingBatch : BOOL
VAR_INPUT
END_VAR
IF NOT Service.AutoMode_SimpleAllocation_Batch.HandShake.Execute 
   AND  NOT Service.AutoMode_AllocateBatchMode_Reverse.HandShake.Execute	THEN
	
	AutoAllocateJobBatch_Ctrl.bSimpleAllocation:=FALSE;
	AutoAllocateJobBatch_Ctrl.bExecute:=Service.AutoMode_AllocateBatchMode.HandShake.Execute;
	AutoAllocateJobBatch_Ctrl.bReset :=Service.AutoMode_AllocateBatchMode.HandShake.Reset;
	AutoAllocateJobBatch_Ctrl.bOccupied:=Service.AutoMode_AllocateBatchMode.HandShake.Occupied;
	AutoAllocateJobBatch_Ctrl.bPause :=Service.AutoMode_AllocateBatchMode.Pause;

	AutoAllocateJobBatch_Ctrl.AutoMode_AllocateMoveBatch.AllocationInfo:=Service.AutoMode_AllocateBatchMode.AllocationInfo;
	AutoAllocateJobBatch_Ctrl.AutoMode_AllocateMoveBatch.NrOfAllocationJob:=Service.AutoMode_AllocateBatchMode.NrOfAllocationJob;

	Service.AutoMode_AllocateBatchMode.WorkedID:=AutoAllocateJobBatch_Ctrl.AutoMode_AllocateMoveBatch.WorkedID;
	Service.AutoMode_AllocateBatchMode.HandShake.Busy:= AutoAllocateJobBatch_Status.bBusy;
	Service.AutoMode_AllocateBatchMode.HandShake.Error:= AutoAllocateJobBatch_Status.bError;
	Service.AutoMode_AllocateBatchMode.HandShake.Done:= AutoAllocateJobBatch_Status.bDone;
	
	RoundBeltMoveJob_Ctrl_Batch :=fb_AllocateBatchMode.RoundBeltMoveJob_Ctrl; 
	RoundBeltMoveJob_Position :=fb_AllocateBatchMode.RoundBeltMoveJob_Position;	
	bAutoAllocateJobDryRun := FALSE;
END_IF
END_METHOD

METHOD PRIVATE M_AutoAllocatingBatch_Reverse : BOOL
VAR_INPUT
END_VAR
	IF NOT Service.AutoMode_AllocateBatchMode.HandShake.Execute 
	   AND NOT Service.AutoMode_SimpleAllocation_Batch.HandShake.Execute THEN
	AutoAllocateJobBatch_Reverse_Ctrl.bExecute:=Service.AutoMode_AllocateBatchMode_Reverse.HandShake.Execute;
	AutoAllocateJobBatch_Reverse_Ctrl.bReset :=Service.AutoMode_AllocateBatchMode_Reverse.HandShake.Reset;
	AutoAllocateJobBatch_Reverse_Ctrl.bOccupied:=Service.AutoMode_AllocateBatchMode_Reverse.HandShake.Occupied;
	AutoAllocateJobBatch_Reverse_Ctrl.bPause :=Service.AutoMode_AllocateBatchMode_Reverse.Pause;

	AutoAllocateJobBatch_Reverse_Ctrl.AutoMode_AllocateMoveBatch.AllocationInfo:=Service.AutoMode_AllocateBatchMode_Reverse.AllocationInfo;
	AutoAllocateJobBatch_Reverse_Ctrl.AutoMode_AllocateMoveBatch.NrOfAllocationJob:=Service.AutoMode_AllocateBatchMode_Reverse.NrOfAllocationJob;

	Service.AutoMode_AllocateBatchMode_Reverse.WorkedID:=AutoAllocateJobBatch_Reverse_Ctrl.AutoMode_AllocateMoveBatch.WorkedID;
	Service.AutoMode_AllocateBatchMode_Reverse.HandShake.Busy:= AutoAllocateJobBatch_Reverse_Status.bBusy;
	Service.AutoMode_AllocateBatchMode_Reverse.HandShake.Error:= AutoAllocateJobBatch_Reverse_Status.bError;
	Service.AutoMode_AllocateBatchMode_Reverse.HandShake.Done:= AutoAllocateJobBatch_Reverse_Status.bDone;
	RoundBeltMoveJob_Ctrl_Batch :=fb_AllocateBatchMode_Reverse.RoundBeltMoveJob_Ctrl; 
	RoundBeltMoveJob_Position :=fb_AllocateBatchMode_Reverse.RoundBeltMoveJob_Position;	

	bAutoAllocateJobDryRun := FALSE;
	
	END_IF
END_METHOD

METHOD PRIVATE M_AutoAllocatingBatch_Simple : BOOL
VAR_INPUT
END_VAR
IF NOT Service.AutoMode_AllocateBatchMode.HandShake.Execute 
   AND NOT Service.AutoMode_AllocateBatchMode_Reverse.HandShake.Execute	THEN
	
	AutoAllocateJobBatch_Ctrl.bSimpleAllocation:=TRUE;
	AutoAllocateJobBatch_Ctrl.bExecute:=Service.AutoMode_SimpleAllocation_Batch.HandShake.Execute;
	AutoAllocateJobBatch_Ctrl.bReset :=Service.AutoMode_SimpleAllocation_Batch.HandShake.Reset;
	AutoAllocateJobBatch_Ctrl.bOccupied:=Service.AutoMode_SimpleAllocation_Batch.HandShake.Occupied;
	AutoAllocateJobBatch_Ctrl.bPause :=Service.AutoMode_SimpleAllocation_Batch.Pause;

	AutoAllocateJobBatch_Ctrl.AutoMode_AllocateMoveBatch.AllocationInfo:=Service.AutoMode_SimpleAllocation_Batch.AllocationInfo;
	AutoAllocateJobBatch_Ctrl.AutoMode_AllocateMoveBatch.NrOfAllocationJob:=Service.AutoMode_SimpleAllocation_Batch.NrOfAllocationJob;

	Service.AutoMode_SimpleAllocation_Batch.WorkedID:=AutoAllocateJobBatch_Ctrl.AutoMode_AllocateMoveBatch.WorkedID;
	Service.AutoMode_SimpleAllocation_Batch.HandShake.Busy:= AutoAllocateJobBatch_Status.bBusy;
	Service.AutoMode_SimpleAllocation_Batch.HandShake.Error:= AutoAllocateJobBatch_Status.bError;
	Service.AutoMode_SimpleAllocation_Batch.HandShake.Done:= AutoAllocateJobBatch_Status.bDone;
	
	RoundBeltMoveJob_Ctrl_Batch :=fb_AllocateBatchMode.RoundBeltMoveJob_Ctrl; 
	RoundBeltMoveJob_Position :=fb_AllocateBatchMode.RoundBeltMoveJob_Position;		

	bAutoAllocateJobDryRun := FALSE;
END_IF
END_METHOD

METHOD PRIVATE M_AutoTurnTable : BOOL
VAR_INPUT
END_VAR
_TurnTableMove.HandShake.Execute:=Service.AutoMode_TurnTableMove.HandShake.Execute;
_TurnTableMove.Position:=Service.AutoMode_TurnTableMove.Position;

Service.AutoMode_TurnTableMove.HandShake.Busy := _TurnTableMove.HandShake.Busy;
Service.AutoMode_TurnTableMove.HandShake.Done := _TurnTableMove.HandShake.Done;
Service.AutoMode_TurnTableMove.HandShake.Error := _TurnTableMove.HandShake.Error;
END_METHOD

METHOD PRIVATE M_CheckAxesHomed : BOOL
VAR_INPUT
END_VAR

VAR 
	AxisIndex : INT;//1-6
	bCheckHome : BOOL:=TRUE;
END_VAR
bCheckHome:=TRUE;

FOR AxisIndex :=1 TO 6 DO
	bCheckHome:=bCheckHome AND	arAxisCtrl_gb[AxisIndex].Admin.Axis.Status.Homed;
END_FOR

M_CheckAxesHomed:=	bCheckHome;
END_METHOD

METHOD M_Clearing
M_StateComplete();
END_METHOD

METHOD M_Complete
M_StateComplete();
END_METHOD

METHOD M_Completing
M_StateComplete();
END_METHOD

METHOD M_Execute
CASE eModeCurrent OF
	E_UnitMode.Manual:
		M_ManualAllocating();
		M_AutoAllocatingBatch_Simple();
		M_AutoAllocatingBatch();
		M_AutoAllocatingBatch_Reverse();
		M_ManualTurnTable();
		M_AutoAllocatingBatch_Reverse();
		//M_TransCVCameraPress_ManualMode();
		//TransCV_Press :=FALSE;

	E_UnitMode.Auto:
	
		M_AutoAllocatingBatch_Simple();
		M_AutoAllocatingBatch();
		M_AutoAllocatingBatch_Reverse();
		M_AutoTurnTable();
		M_TransCVCameraPress();
END_CASE
//M_StateComplete();
A00_Service();
A01_RoundBeltAccessControl();
A02_PulloutAccessControl();
//bHomed :=M_CheckAxesHomed();
END_METHOD

METHOD PUBLIC M_GetPulloutAccess : BOOL
VAR_INPUT
	 ControlAccess:	 E_RoundBeltControlAccess;
END_VAR
IF THIS^.PulloutControlAccess = E_RoundBeltControlAccess.Host AND 
	NOT (fbPulloutCV.Execute OR fbPulloutCV.Busy OR fbPulloutCV.Done) THEN
	THIS^.PulloutControlAccess := ControlAccess;
	M_GetPulloutAccess := TRUE;
 ELSE
	M_GetPulloutAccess := FALSE;	
 END_IF
END_METHOD

METHOD PUBLIC M_GetRoundBeltAccess : BOOL
VAR_INPUT
	 ControlAccess:	 E_RoundBeltControlAccess;
END_VAR
IF THIS^.RoundBeltControlAccess = E_RoundBeltControlAccess.Host AND 
	NOT (RoundBeltControl.xExecute OR RoundBeltControl.xBusy OR RoundBeltControl.xDone) THEN
	THIS^.RoundBeltControlAccess := ControlAccess;
	M_GetRoundBeltAccess := TRUE;
 ELSE
	M_GetRoundBeltAccess := FALSE;	
 END_IF
END_METHOD

METHOD M_Held
M_StateComplete();
END_METHOD

METHOD M_Holding
M_StateComplete();
END_METHOD

METHOD M_Idle
M_StateComplete();
END_METHOD

METHOD M_InactiveRoundBeltInternalCtrl : BOOL
VAR_INPUT
END_VAR
bReloadRotateBeltRequest := FALSE;

M_InactiveRoundBeltInternalCtrl := true; // Method end
END_METHOD

METHOD PRIVATE M_ManualAllocating : BOOL
VAR_INPUT
END_VAR

VAR_INST 
	
END_VAR

	AutoAllocateJobBatch_Ctrl.bSimpleAllocation:=FALSE;
	AutoAllocateJobBatch_Ctrl.bReset:=Service.AllocateMoveStructure.HandShake.Reset;
	AutoAllocateJobBatch_Ctrl.bPause:=FALSE;
	AutoAllocateJobBatch_Ctrl.bOccupied :=Service.AllocateMoveStructure.HandShake.Occupied;
	AutoAllocateJobBatch_Ctrl.bExecute:=Service.AllocateMoveStructure.HandShake.Execute;
	AutoAllocateJobBatch_Ctrl.AutoMode_AllocateMoveBatch.NrOfAllocationJob:=1;
	AutoAllocateJobBatch_Ctrl.AutoMode_AllocateMoveBatch.AllocationInfo[0].FastMode:=FALSE;
	AutoAllocateJobBatch_Ctrl.AutoMode_AllocateMoveBatch.AllocationInfo[0].SyncMode:=FALSE	;
	
	AutoAllocateJobBatch_Ctrl.AutoMode_AllocateMoveBatch.AllocationInfo[0].PickingNeedleInfo[0].CycleStart:=TRUE;
	AutoAllocateJobBatch_Ctrl.AutoMode_AllocateMoveBatch.AllocationInfo[0].PickingNeedleInfo[0].Box:=LREAL_TO_UINT( Service.AllocateMoveStructure.Frombox);
	AutoAllocateJobBatch_Ctrl.AutoMode_AllocateMoveBatch.AllocationInfo[0].PickingNeedleInfo[0].Clip:=LREAL_TO_INT(Service.AllocateMoveStructure.Clip);
	AutoAllocateJobBatch_Ctrl.AutoMode_AllocateMoveBatch.AllocationInfo[0].PickingNeedleInfo[0].NeedleLocation:=LREAL_TO_INT(Service.AllocateMoveStructure.FromPosition);
	AutoAllocateJobBatch_Ctrl.AutoMode_AllocateMoveBatch.AllocationInfo[0].PlacingNeedleInfo[0].CycleStart:=TRUE;
	
	AutoAllocateJobBatch_Ctrl.AutoMode_AllocateMoveBatch.AllocationInfo[0].PlacingNeedleInfo[0].Box :=LREAL_TO_UINT(Service.AllocateMoveStructure.Tobox);
	AutoAllocateJobBatch_Ctrl.AutoMode_AllocateMoveBatch.AllocationInfo[0].PlacingNeedleInfo[0].Clip:=LREAL_TO_INT(Service.AllocateMoveStructure.Clip);
	AutoAllocateJobBatch_Ctrl.AutoMode_AllocateMoveBatch.AllocationInfo[0].PlacingNeedleInfo[0].NeedleLocation :=LREAL_TO_INT(Service.AllocateMoveStructure.ToPosition);

	Service.AllocateMoveStructure.HandShake.Busy :=AutoAllocateJobBatch_Status.bBusy;
	Service.AllocateMoveStructure.HandShake.Done :=AutoAllocateJobBatch_Status.bDone;
	Service.AllocateMoveStructure.HandShake.Error :=AutoAllocateJobBatch_Status.bError;
	bAutoAllocateJobDryRun := TRUE;
END_METHOD

METHOD PRIVATE M_ManualTurnTable : BOOL
VAR_INPUT
END_VAR
_TurnTableMove.HandShake.Execute:=Service.TurnTableMove.HandShake.Execute;
_TurnTableMove.Position:=Service.TurnTableMove.Position;

Service.TurnTableMove.HandShake.Busy := _TurnTableMove.HandShake.Busy;
Service.TurnTableMove.HandShake.Done := _TurnTableMove.HandShake.Done;
Service.TurnTableMove.HandShake.Error := _TurnTableMove.HandShake.Error;
END_METHOD

METHOD PUBLIC M_ReleasePulloutAccess : BOOL
VAR_INPUT
 ControlAccess:	 E_RoundBeltControlAccess;
END_VAR
IF ControlAccess = THIS^.PulloutControlAccess THEN
		THIS^.PulloutControlAccess := E_RoundBeltControlAccess.Host;
		M_ReleasePulloutAccess := TRUE;
	ELSE
		M_ReleasePulloutAccess := FALSE;
	
END_IF
END_METHOD

METHOD PUBLIC M_ReleaseRoundBeltAccess : BOOL
VAR_INPUT
 ControlAccess:	 E_RoundBeltControlAccess;
END_VAR
IF ControlAccess = THIS^.RoundBeltControlAccess THEN
		THIS^.RoundBeltControlAccess := E_RoundBeltControlAccess.Host;
		M_ReleaseRoundBeltAccess := TRUE;
	ELSE
		M_ReleaseRoundBeltAccess := FALSE;
	
END_IF
END_METHOD

METHOD M_ResetReloadRoundBeltAction : BOOL
VAR_INPUT
END_VAR
RoundBeltMoveJob_Ctrl.Execute := FALSE;

M_ResetReloadRoundBeltAction := true; // Method end
END_METHOD

METHOD M_Resetting
IF __ISVALIDREF(Cylinder) THEN
	Clip.stCylinders.Cylinder0 REF= Cylinder.List.fbAllocateRobot_LeftClamp1;
	Clip.stCylinders.Cylinder1 REF= Cylinder.List.fbAllocateRobot_LeftClamp2;
	Clip.stCylinders.Cylinder2 REF= Cylinder.List.fbAllocateRobot_RightClamp1;
	Clip.stCylinders.Cylinder3 REF= Cylinder.List.fbAllocateRobot_RightClamp2;
	Cylinders.stCylinders.Cylinder0 REF= Cylinder.List.fbAllocateRobot_LeftVert1;
	Cylinders.stCylinders.Cylinder1 REF= Cylinder.List.fbAllocateRobot_LeftVert2;
	Cylinders.stCylinders.Cylinder2 REF= Cylinder.List.fbAllocateRobot_RightVert1;
	Cylinders.stCylinders.Cylinder3 REF= Cylinder.List.fbAllocateRobot_RightVert2;	
END_IF

M_StateComplete();
END_METHOD

METHOD PUBLIC M_StartAllocatePulloutAction : BOOL
VAR_INPUT
	CV_ForwardTime :TIME;
	CV_BackwardTIme : TIME;
	CommandType : E_PullOutConveyorCommandType; // Select PullOut conveyor command.
END_VAR
AutoPullout_Internal_Ctrl.Execute := TRUE;
AutoPullout_Internal_Info.ConveyorReverseTime := CV_BackwardTIme;
AutoPullout_Internal_Info.ConveyorRunningTime := CV_ForwardTime;
AutoPullout_Internal_Info.CommandType := CommandType;
M_StartAllocatePulloutAction := TRUE; // Method end
END_METHOD

METHOD M_StartHoming
VAR_INPUT
END_VAR
fbAllocateHome.xExecute := true;
END_METHOD

METHOD M_Starting
M_StateComplete();
END_METHOD

(* This Method is used to start round belt action : unlock pin and move to target position
	also injection the action parameter.
*)
METHOD M_StartReloadRoundBeltAtion : BOOL
VAR_INPUT
	ReloadStation : E_RoundBeltStation;
END_VAR
VAR_INST
	_ReloadStation : E_RoundBeltStation;
END_VAR
IF (ReloadStation > 12) THEN
	_ReloadStation := (ReloadStation -12 );
//	_ReloadStation := (ReloadStation -6 );
ELSE
	_ReloadStation := ReloadStation + 28;
END_IF
IF F_Even(_ReloadStation) THEN
	_ReloadStation := _ReloadStation-1;
END_IF

//IF ReloadStation > 6 THEN
//	_ReloadStation := ReloadStation -6;
//ELSE
//	_ReloadStation := ReloadStation +14;
//END_IF
//AutoRotatebelt_Internal_Ctrl.uiLatch := E_Pistons.LoadingBoxRegion;
//AutoRotatebelt_Internal_Ctrl.uiStation :=  _ReloadStation;
//AutoRotatebelt_Internal_Ctrl.Timeout := T#15S;
//AutoRotatebelt_Internal_Ctrl.bSendPressBox := FALSE; // Release allocate zone, press box cylinder in backward position
RoundBeltMoveJob_Position_FanucRobot := _ReloadStation;
RoundBeltMoveJob_Ctrl.Execute := TRUE;

M_StartReloadRoundBeltAtion := TRUE; // Method end
END_METHOD

METHOD M_StartStoragePulloutAction : BOOL
VAR_INPUT
	CV_ForwardTime :TIME;
	CV_BackwardTIme : TIME;
	CommandType : E_PullOutConveyorCommandType; // Select PullOut conveyor command.
END_VAR
RobotPullout_Internal_Ctrl.Execute := TRUE;
RobotPullout_Internal_Info.CommandType := CommandType;
RobotPullout_Internal_Info.ConveyorReverseTime := CV_BackwardTIme;
RobotPullout_Internal_Info.ConveyorRunningTime := CV_ForwardTime;
M_StartStoragePulloutAction := TRUE; // Method end
END_METHOD

METHOD M_StopAllocatePulloutAction : BOOL
VAR_INPUT
END_VAR
AutoPullout_Internal_Ctrl.Execute := FALSE;
M_StopAllocatePulloutAction := TRUE; // Methode end
END_METHOD

METHOD M_StopHoming
VAR_INPUT
END_VAR
fbAllocateHome.xExecute := False;
END_METHOD

METHOD M_Stopped
M_StateComplete();
END_METHOD

METHOD M_Stopping
M_StateComplete();
END_METHOD

METHOD M_StopStoragePulloutAction : BOOL
VAR_INPUT
END_VAR
RobotPullout_Internal_Ctrl.Execute := FALSE;
M_StopStoragePulloutAction := TRUE; //Method End
END_METHOD

METHOD M_Suspended
M_StateComplete();
END_METHOD

METHOD M_Suspending
M_StateComplete();
END_METHOD

METHOD PUBLIC M_TransCVCameraPress : BOOL
VAR_INPUT
END_VAR
VAR_INST
	
END_VAR
IF NOT TransCV_Press THEN
	Cylinder.List.fbSameSizeCV_Press2.M_Extend();
	Cylinder.List.fbDifferentSizeCV_Press1.M_Extend();
	TransCV_Press:=true;
END_IF
END_METHOD

METHOD PUBLIC M_TransCVCameraPress_ManualMode : BOOL
VAR_INPUT
END_VAR
IF TransCV_Press THEN
TransCV_Press := FALSE;
Cylinder.List.fbSameSizeCV_Press2.M_Retract();
Cylinder.List.fbDifferentSizeCV_Press1.M_Retract();
END_IF
END_METHOD

METHOD M_Undefined
M_StateComplete();
END_METHOD

METHOD M_Unholding
M_StateComplete();
END_METHOD

METHOD M_Unsuspending
M_StateComplete();
END_METHOD

END_FUNCTION_BLOCK

// ---- Library/20_MachineUnits/22_AllocateArea/Service/FB_AllocateAreaHome.TcPOU
FUNCTION_BLOCK FB_AllocateAreaHome EXTENDS FB_ActionBasic
VAR_INPUT
    xExecute      : BOOL;
    xAbort        : BOOL;

    Cylinder : REFERENCE TO UNI_CylinderList;
	Motor    : REFERENCE TO UNI_MotorList;
	CurrentData      : ST_SetupPara;
    TimeOut  : LREAL := 90; // Unit : s
	Homed : REFERENCE TO BOOL;
END_VAR
VAR_OUTPUT
    xAborted : BOOL;
    iErrorID : INT;
    ErrorMsg : STRING;
	AxisHomingRequest : BOOL;
END_VAR
VAR
    StateBehavior   : CBML.ETrigATo;
    CurrentPosition : ST_PositionTable;
    uiCyclicStep    : UINT := 0;
    uiIndexLoop     : UINT;
	fbExecuteEdgeDetect :FB_EdgeDetect;
END_VAR

THIS^.IBehaviourModel := StateBehavior;
StateBehavior(xExecute := xExecute,
              xAbort := xAbort OR fbExecuteEdgeDetect.xFallingEdge,
              udiTimeOut := LREAL_TO_UDINT( TimeOut*1000000),
              xDone => xDone,
              xBusy => xBusy,
              xError => xError,
              xAborted => xAborted);	

//Make sure that C# turns off execute to shut down the service
fbExecuteEdgeDetect(xInput :=xExecute);

//Error Msg
iErrorID := StateBehavior._model.iErrorID;
ErrorMsg := M_GetErrorMsg(xErrorID := iErrorID);

METHOD CleanupAction
VAR_INPUT
    xAbortProposed : BOOL;
    iErrorIDProposed: INT;
END_VAR
VAR_OUTPUT
    xComplete : BOOL := TRUE;
    xAbort: BOOL := xAbortProposed;
 	iErrorID : INT := iErrorIDProposed;
END_VAR
uiCyclicStep := 0;
END_METHOD

METHOD CyclicAction
VAR_INPUT
    itfTimingController : CBML.ITimingController;
END_VAR
VAR_OUTPUT
    xComplete : BOOL := TRUE;
    iErrorID : INT := 0;
END_VAR
VAR_INST
	
END_VAR

VAR
	AxisIndex 		: INT ; //1-6
	CylinderIndex 	: INT ;
	MotorIndex		: INT ;// 23-26
	bAxesCheck 		: BOOL;
	bCylinderCheck  : BOOL;
	bHomeCheck 		: BOOL;
	bMotorCheck		: BOOL;
END_VAR
xComplete := FALSE;
CASE uiCyclicStep OF
    0: //Check Motor
		bMotorCheck:= TRUE;
		FOR MotorIndex :=23 TO 26 DO
			bMotorCheck := bMotorCheck AND Motor.arMotor[MotorIndex].InStopped;
			IF Motor.arMotor[MotorIndex].xError THEN
				Motor.arMotor[MotorIndex].M_Reset();
			ELSE
				Motor.arMotor[MotorIndex].M_MotorStop();
			END_IF
		END_FOR
		IF bMotorCheck THEN
			uiCyclicStep:=100;
		END_IF
		
	100: // Check Axes error
		bAxesCheck:=TRUE;
		FOR AxisIndex :=1 TO 6 DO
			bAxesCheck := bAxesCheck AND NOT arAxisCtrl_gb[AxisIndex].Admin.Axis.Status.Error;
			IF arAxisCtrl_gb[AxisIndex].Admin.Axis.Status.Error THEN
				arAxisCtrl_gb[AxisIndex].Admin.ClearError:=TRUE;
			END_IF
		END_FOR
		
		IF bAxesCheck THEN
			uiCyclicStep:=200;
		END_IF
			
	200: // Reset All cylinder
		FOR AxisIndex :=1 TO 6 DO 	arAxisCtrl_gb[AxisIndex].Admin.ClearError:=FALSE;	END_FOR
		bCylinderCheck:=TRUE;
		FOR CylinderIndex:=15 TO 20 DO
			bCylinderCheck:=bCylinderCheck AND NOT Cylinder.arCylinder[CylinderIndex].xError;
			IF Cylinder.arCylinder[CylinderIndex].xError THEN
				Cylinder.arCylinder[CylinderIndex].M_Reset();
			END_IF
		END_FOR
		FOR CylinderIndex:=27 TO 53 DO
			bCylinderCheck:=bCylinderCheck AND NOT Cylinder.arCylinder[CylinderIndex].xError;
			IF Cylinder.arCylinder[CylinderIndex].xError THEN
				Cylinder.arCylinder[CylinderIndex].M_Reset();
			END_IF
		END_FOR
		IF bCylinderCheck THEN
			uiCyclicStep:=300;
		END_IF
		
	300:
		bCylinderCheck:=TRUE;
		FOR CylinderIndex:=15 TO 20 DO
			bCylinderCheck:=bCylinderCheck AND Cylinder.arCylinder[CylinderIndex].InRearPosition;
			Cylinder.arCylinder[CylinderIndex].M_Retract();			
		END_FOR
		FOR CylinderIndex:=27 TO 53 DO
			bCylinderCheck:=bCylinderCheck AND Cylinder.arCylinder[CylinderIndex].InRearPosition;
			Cylinder.arCylinder[CylinderIndex].M_Retract();			
		END_FOR
		IF bCylinderCheck THEN
			uiCyclicStep:=400;
		END_IF

	400:
		//bHomeCheck := TRUE;
		//IF DAS_CoreSys.MachineControl.fanucrobot.List.StorageRobot._uo1.UO07_AtPerch THEN
			AxisHomingRequest := TRUE;
			IF NOT arAxisCtrl_gb[AxisNo.TurnTable].Admin.Axis.Status.Homed  THEN
			uiCyclicStep:=500;
		//END_IF
		END_IF
		
		

500:	
		bHomeCheck:=TRUE;
		FOR AxisIndex :=1 TO 6 DO
			bHomeCheck := bHomeCheck AND arAxisStatus_gb[AxisIndex].Admin.CmdDone ;//AND arAxisCtrl_gb[AxisIndex].Admin.Axis.Status.Homed;
		END_FOR
		bHomeCheck := arAxisCtrl_gb[AxisNo.Allocate_X].Admin.Axis.Status.Homed AND
			 arAxisCtrl_gb[AxisNo.OutRobot_X].Admin.Axis.Status.Homed AND 
			 arAxisCtrl_gb[AxisNo.OutRobot_Y].Admin.Axis.Status.Homed AND 
			 arAxisCtrl_gb[AxisNo.RoundBelt].Admin.Axis.Status.Homed AND 
			 arAxisCtrl_gb[AxisNo.TurnTable].Admin.Axis.Status.Homed AND 
			 GVL_Machine.AllocatYAxisHome;

		
		IF bHomeCheck THEN
			uiCyclicStep:=600;
		END_IF
	
	600:
		Homed := TRUE;
		xComplete := TRUE;
END_CASE
END_METHOD

METHOD ExitAction
VAR_INPUT
    xAfterCleanup : BOOL;
    xInCopyCode : BOOL;
END_VAR
END_METHOD

METHOD M_GetErrorMsg : T_MaxString
VAR_INPUT
	xErrorID: INT;
END_VAR

VAR
	
END_VAR
CASE xErrorID OF
	0:
		M_GetErrorMsg := 'No Error';
	1:
		M_GetErrorMsg := 'Action time out';
//	2:
//		M_GetErrorMsg := 'Position Data invalid';
//	3:
//		M_GetErrorMsg := 'Index invalid';
//	4:
//		M_GetErrorMsg := 'Axis roundbelt not ready has Error';
//	5:
//		M_GetErrorMsg := 'Cylinder not ready has Error';
//	6:
//		M_GetErrorMsg := 'Axis RoundBelt has Error';
//	7:
//		M_GetErrorMsg := 'ChargeZone_Plug has Error';
//	8:
//		M_GetErrorMsg := 'TransmitCVZone_Plug has Error';
//	9:
//		M_GetErrorMsg := 'WorkZone_Plug has Error';
//	10:
//		M_GetErrorMsg := 'WorkZone_Press has Error';
END_CASE
END_METHOD

METHOD PRIVATE M_SetAllHomePars : BOOL
VAR_INPUT
END_VAR
//Allocate X

arAxisCtrl_gb[AxisNo.Allocate_X].Admin._OpMode.en := ModeHoming;

//Allocate Y
arAxisCtrl_gb[AxisNo.Allocate_Y].Admin._OpMode.en := ModePosAbs;

//OutRobot X
arAxisCtrl_gb[AxisNo.OutRobot_X].Admin._OpMode.en := ModeHoming;

//OutRobot Y

arAxisCtrl_gb[AxisNo.OutRobot_Y].Admin._OpMode.en := ModeHoming;

//RoundBelt

arAxisCtrl_gb[AxisNo.RoundBelt].Admin._OpMode.en := ModeHoming;

//TurnTable

arAxisCtrl_gb[AxisNo.TurnTable].Admin._OpMode.en := ModeHoming;
END_METHOD

METHOD ResetAction
VAR_OUTPUT
    xComplete : BOOL := TRUE;
END_VAR
AxisHomingRequest := FALSE;
uiCyclicStep := 0;
END_METHOD

METHOD StartAction
VAR_OUTPUT
    xComplete : BOOL := TRUE;
	iErrorID : INT := 0;
END_VAR
xComplete := FALSE;

uiCyclicStep := 0;
Homed := FALSE;

xComplete := TRUE;
END_METHOD

END_FUNCTION_BLOCK

// ---- Library/99_Utilities/FB_EdgeDetect.TcPOU
FUNCTION_BLOCK FB_EdgeDetect
VAR_INPUT
    xInput      : BOOL;     // 監視的布林輸入
END_VAR

VAR_OUTPUT
    xRisingEdge : BOOL;     // 上升沿輸出 (R_Trig)
    xFallingEdge: BOOL;     // 下降沿輸出 (F_Trig)
END_VAR

VAR
    xLastInput  : BOOL;     // 前一個週期的輸入狀態
END_VAR

// 程式邏輯
// 檢測上升沿 (FALSE -> TRUE)
xRisingEdge := xInput AND NOT xLastInput;

// 檢測下降沿 (TRUE -> FALSE)
xFallingEdge := NOT xInput AND xLastInput;

// 儲存當前輸入狀態供下一個週期使用
xLastInput := xInput;

END_FUNCTION_BLOCK

// ---- Library/20_MachineUnits/22_AllocateArea/Service/FB_RoundBeltService.TcPOU
FUNCTION_BLOCK FB_RoundBeltService EXTENDS FB_ActionBasic
VAR_INPUT
    xExecute      : BOOL;
    xAbort        : BOOL;
    TargetStation : INT;

    Cylinder : REFERENCE TO UNI_CylinderList;
    TimeOut  : LREAL := 90; // Unit : s
END_VAR
VAR_OUTPUT
    xAborted : BOOL;
    iErrorID : INT;
    ErrorMsg : STRING;
END_VAR
VAR
    StateBehavior   : CBML.ETrigATo;
    CurrentPosition : ST_PositionTable;
    CurrentData     : ARRAY[1..21] OF ST_PositionTable;
    uiCyclicStep    : UINT := 0;
    uiIndexLoop     : UINT;
	fbExecuteEdgeDetect :FB_EdgeDetect;
END_VAR

THIS^.IBehaviourModel := StateBehavior;
StateBehavior(xExecute := xExecute,
              xAbort := xAbort OR fbExecuteEdgeDetect.xFallingEdge,
              udiTimeOut := LREAL_TO_UDINT( TimeOut*1000000),
              xDone => xDone,
              xBusy => xBusy,
              xError => xError,
              xAborted => xAborted);

//Make sure that C# turns off execute to shut down the service
fbExecuteEdgeDetect(xInput :=xExecute);

//Error Msg
iErrorID := StateBehavior._model.iErrorID;
ErrorMsg := M_GetErrorMsg(xErrorID := iErrorID);

			  
A00_ReadPositionData();

ACTION A00_ReadPositionData:
FOR uiIndexLoop := 1 TO 20 DO
    CurrentData[uiIndexLoop] := FUN_GetPositionTableData(PositionName := 'B', Index := UINT_TO_LREAL(uiIndexLoop), Clip := E_ClipNo.A);
END_FOR
END_ACTION

METHOD CleanupAction
VAR_INPUT
    xAbortProposed : BOOL;
    iErrorIDProposed: INT;
END_VAR
VAR_OUTPUT
    xComplete : BOOL := TRUE;
    xAbort: BOOL := xAbortProposed;
 	iErrorID : INT := iErrorIDProposed;
END_VAR
uiCyclicStep := 0;
END_METHOD

METHOD CyclicAction
VAR_INPUT
    itfTimingController : CBML.ITimingController;
END_VAR
VAR_OUTPUT
    xComplete : BOOL := TRUE;
    iErrorID : INT := 0;
END_VAR
VAR_INST
	
END_VAR
xComplete := FALSE;
CASE uiCyclicStep OF
    0:
		//Check if current station is same as target
		IF ABS(CurrentPosition.X_Pos -  arAxisCtrl_gb[AxisNo.RoundBelt].Admin.Axis.NcToPlc.ModuloSetPos) < 0.2 THEN
			uiCyclicStep := 200;
			ELSE
			uiCyclicStep := 50;	
		END_IF
	50:
		// Retract all cylinders
        Cylinder.List.fbRoundBelt_ChargeZone_Plug.M_Retract();
        Cylinder.List.fbRoundBelt_TransmitCVZone_Plug.M_Retract();
        Cylinder.List.fbRoundBelt_WorkZone_Plug.M_Retract();
        Cylinder.List.fbRoundBelt_WorkZone_Press.M_Retract();

        IF Cylinder.List.fbRoundBelt_ChargeZone_Plug.InRearPosition AND
            Cylinder.List.fbRoundBelt_TransmitCVZone_Plug.InRearPosition AND
            Cylinder.List.fbRoundBelt_WorkZone_Plug.InRearPosition AND
            Cylinder.List.fbRoundBelt_WorkZone_Press.InRearPosition THEN
            uiCyclicStep := 100;
        END_IF
    100: 
	    // Move round belt to target station
        arAxisCtrl_gb[AxisNo.RoundBelt].PosMode.Position := CurrentPosition.X_Pos;
		 IF  arAxisCtrl_gb[AxisNo.RoundBelt].Admin.Axis.Status.Moving THEN
				uiCyclicStep := 190;
		 END_IF
		
	190:
        IF arAxisStatus_gb[AxisNo.RoundBelt].Admin._OpModeAck = ModePosAbs AND arAxisStatus_gb[AxisNo.RoundBelt].Admin.CmdDone AND
			(arAxisCtrl_gb[AxisNo.RoundBelt].Admin.Axis.Status.InTargetPosition OR arAxisCtrl_gb[AxisNo.RoundBelt].Admin.Axis.Status.Operational)
		THEN
            uiCyclicStep := 200;
        END_IF
	200:
        Cylinder.List.fbRoundBelt_ChargeZone_Plug.M_Extend();
        Cylinder.List.fbRoundBelt_TransmitCVZone_Plug.M_Extend();
        Cylinder.List.fbRoundBelt_WorkZone_Plug.M_Extend();
        

        IF Cylinder.List.fbRoundBelt_ChargeZone_Plug.InFrontPosition AND
            Cylinder.List.fbRoundBelt_TransmitCVZone_Plug.InFrontPosition AND
            Cylinder.List.fbRoundBelt_WorkZone_Plug.InFrontPosition THEN
            uiCyclicStep := 300;
        END_IF
	300:
		Cylinder.List.fbRoundBelt_WorkZone_Press.M_Extend();
		IF  Cylinder.List.fbRoundBelt_WorkZone_Press.InFrontPosition THEN
            xComplete := TRUE;
        END_IF
		//	xComplete := TRUE;
END_CASE

IF arAxisCtrl_gb[AxisNo.RoundBelt].Admin.Axis.Status.Error THEN
    iErrorID := 6; // Axis RoundBelt has error
END_IF

IF Cylinder.List.fbRoundBelt_ChargeZone_Plug.xError THEN
    iErrorID := 7;
END_IF

IF Cylinder.List.fbRoundBelt_TransmitCVZone_Plug.xError THEN
    iErrorID := 8;
END_IF

IF Cylinder.List.fbRoundBelt_WorkZone_Plug.xError THEN
    iErrorID := 9;
END_IF

IF Cylinder.List.fbRoundBelt_WorkZone_Press.xError THEN
    iErrorID := 10;
END_IF
END_METHOD

METHOD ExitAction
VAR_INPUT
    xAfterCleanup : BOOL;
    xInCopyCode : BOOL;
END_VAR
END_METHOD

METHOD M_GetErrorMsg : T_MaxString
VAR_INPUT
	xErrorID: INT;
END_VAR

VAR
	
END_VAR
CASE xErrorID OF
	0:
		M_GetErrorMsg := 'No Error';
	1:
		M_GetErrorMsg := 'Action time out';
	2:
		M_GetErrorMsg := 'Position Data invalid';
	3:
		M_GetErrorMsg := 'Index invalid';
	4:
		M_GetErrorMsg := 'Axis roundbelt not ready has Error';
	5:
		M_GetErrorMsg := 'Cylinder not ready has Error';
	6:
		M_GetErrorMsg := 'Axis RoundBelt has Error';
	7:
		M_GetErrorMsg := 'ChargeZone_Plug has Error';
	8:
		M_GetErrorMsg := 'TransmitCVZone_Plug has Error';
	9:
		M_GetErrorMsg := 'WorkZone_Plug has Error';
	10:
		M_GetErrorMsg := 'WorkZone_Press has Error';
END_CASE
END_METHOD

